ExpectedCount := 0;
ActualCount	  := Sink.LinesWritten;
Test.AssertEqual(ExpectedCount, ActualCount, 'nothing was written');

// Seen but not narrated - the distinction that makes the quiet default safe.
ExpectedCount := 2;
ActualCount	  := Sink.TestsSeen;
Test.AssertEqual(ExpectedCount, ActualCount, 'but both were seen');
Run := TRUE;
END_METHOD

END_FUNCTION_BLOCK

// ---- Tests/LogReporter/TEST_LogReporterWritesFailuresAndErrors.TcPOU
// A failure is an error: the code under test was shown to be wrong. An error is a

// warning: the test could not run, so nothing was shown about the code at all.

//

// Counted apart because a build should react differently to each.//

// WHAT THIS CANNOT CHECK: whether the line actually reached the TwinCAT log, or

// what it says. ADSLOGSTR gives no answer back. The counters prove which BRANCH

// was taken; the wording has to be read once, by eye, in the Logged Events window.

// Saying so is better than a test that implies more than it establishes.
FUNCTION_BLOCK TEST_LogReporterWritesFailuresAndErrors IMPLEMENTS I_Test
VAR
	Sink		  : TestLogReporter;
	ExpectedCount : UDINT;
	ActualCount	  : UDINT;
END_VAR

METHOD Run : BOOL
VAR_INPUT
	Enable : BOOL;
	Test   : I_TestAssertions;
END_VAR
Sink.TestFinished(SuiteLabel	:= 'suite',
				  TestLabel		:= 'a failure',
				  Location		:= '',
				  Status		:= E_TestStatus.Failed,
				  Kind			:= E_FailureKind.ValueMismatch,
				  Summary		:= 'expected 1, actual 2',
				  ElapsedTime	:= 0.0,
				  ElapsedCycles := 1,
				  Assertions	:= 1);

Sink.TestFinished(SuiteLabel	:= 'suite',
				  TestLabel		:= 'an error',
				  Location		:= '',
				  Status		:= E_TestStatus.Errored,
				  Kind			:= E_FailureKind.Environment,
				  Summary		:= 'the axis would not power',
				  ElapsedTime	:= 0.0,
				  ElapsedCycles := 1,
				  Assertions	:= 1);

ExpectedCount := 1;
ActualCount	  := Sink.FailuresLogged;
Test.AssertEqual(ExpectedCount, ActualCount, 'the failure was logged');
ActualCount := Sink.ErrorsLogged;
Test.AssertEqual(ExpectedCount, ActualCount, 'the error was logged separately');
ExpectedCount := 2;
ActualCount	  := Sink.LinesWritten;
Test.AssertEqual(ExpectedCount, ActualCount, 'two lines, not one and not three');
Run := TRUE;
END_METHOD

END_FUNCTION_BLOCK

// ---- Tests/LogReporter/TEST_LogReporterNarratesWhenAsked.TcPOU
// SetVerbosity(TRUE) turns the narration back on, for a rig where the log IS the

// artifact and a passing test that stops appearing is the signal.//

// WHAT THIS CANNOT CHECK: whether the line actually reached the TwinCAT log, or

// what it says. ADSLOGSTR gives no answer back. The counters prove which BRANCH

// was taken; the wording has to be read once, by eye, in the Logged Events window.

// Saying so is better than a test that implies more than it establishes.
FUNCTION_BLOCK TEST_LogReporterNarratesWhenAsked IMPLEMENTS I_Test
VAR
	Sink		  : TestLogReporter;
	ExpectedCount : UDINT;
	ActualCount	  : UDINT;
END_VAR

METHOD Run : BOOL
VAR_INPUT
	Enable : BOOL;
	Test   : I_TestAssertions;
END_VAR
Sink.SetVerbosity(TRUE);
Sink.TestFinished(SuiteLabel	:= 'suite',
				  TestLabel		:= 'a pass',
				  Location		:= '',
				  Status		:= E_TestStatus.Passed,
				  Kind			:= E_FailureKind.None,
				  Summary		:= '',
				  ElapsedTime	:= 0.0,
				  ElapsedCycles := 1,
				  Assertions	:= 1);

ExpectedCount := 1;
ActualCount	  := Sink.LinesWritten;
Test.AssertEqual(ExpectedCount, ActualCount, 'the pass was narrated');

// And it can be turned off again.
Sink.SetVerbosity(FALSE);
Sink.TestFinished(SuiteLabel	:= 'suite',
				  TestLabel		:= 'another pass',
				  Location		:= '',
				  Status		:= E_TestStatus.Passed,
				  Kind			:= E_FailureKind.None,
				  Summary		:= '',
				  ElapsedTime	:= 0.0,
				  ElapsedCycles := 1,
				  Assertions	:= 1);

ActualCount := Sink.LinesWritten;
Test.AssertEqual(ExpectedCount, ActualCount, 'and quiet again afterwards');
Run := TRUE;
END_METHOD

END_FUNCTION_BLOCK

// ---- Tests/LogReporter/TEST_LogReporterAlwaysWritesFrameworkErrors.TcPOU
// A framework error is never silent and is never affected by verbosity. It is the

// framework saying it could not do something - a rejected registration, a teardown

// that overran - and none of those is a test result that can be suppressed.//

// WHAT THIS CANNOT CHECK: whether the line actually reached the TwinCAT log, or

// what it says. ADSLOGSTR gives no answer back. The counters prove which BRANCH

// was taken; the wording has to be read once, by eye, in the Logged Events window.

// Saying so is better than a test that implies more than it establishes.
FUNCTION_BLOCK TEST_LogReporterAlwaysWritesFrameworkErrors IMPLEMENTS I_Test
VAR
	Sink		  : TestLogReporter;
	Fanout		  : TestReporterFanout;
	Attached	  : BOOL;
	ExpectedCount : UDINT;
	ActualCount	  : UDINT;
END_VAR

METHOD Run : BOOL
VAR_INPUT
	Enable : BOOL;
	Test   : I_TestAssertions;
END_VAR
// Quiet mode is the default, and must not silence this.
Sink.FrameworkError(Source := 'a suite', Message := 'registration was rejected');
ExpectedCount := 1;
ActualCount	  := Sink.FrameworkErrorsLogged;
Test.AssertEqual(ExpectedCount, ActualCount, 'logged despite the quiet default');
ActualCount := Sink.LinesWritten;
Test.AssertEqual(ExpectedCount, ActualCount, 'and it produced a line');

// It is a real I_TestReporter, so the fan-out takes it like any other sink.
Attached := Fanout.Attach(Sink);
Test.AssertTrue(Attached, 'the fan-out accepts it');
Fanout.FrameworkError(Source := 'a suite', Message := 'through the fan-out');
ExpectedCount := 2;
ActualCount	  := Sink.FrameworkErrorsLogged;
Test.AssertEqual(ExpectedCount, ActualCount, 'and reaches it that way too');

// Nothing asynchronous, so it never holds a run open.
Test.AssertTrue(Sink.IsIdle, 'the log sink is always idle');
Test.AssertTrue(Fanout.IsIdle, 'so the fan-out is too');
Run := TRUE;
END_METHOD

END_FUNCTION_BLOCK

// ---- Tests/LogReporter/TEST_LogReporterSummarisesASuite.TcPOU
// One line per suite, carrying the counts, with severity following the outcome -

// so a log filtered to errors still shows WHICH suite was responsible rather than

// only the individual failures.//

// WHAT THIS CANNOT CHECK: whether the line actually reached the TwinCAT log, or

// what it says. ADSLOGSTR gives no answer back. The counters prove which BRANCH

// was taken; the wording has to be read once, by eye, in the Logged Events window.

// Saying so is better than a test that implies more than it establishes.
FUNCTION_BLOCK TEST_LogReporterSummarisesASuite IMPLEMENTS I_Test
VAR
	Sink		  : TestLogReporter;
	Tally		  : TestRunTally;
	ExpectedCount : UDINT;
	ActualCount	  : UDINT;
END_VAR

METHOD Run : BOOL
VAR_INPUT
	Enable : BOOL;
	Test   : I_TestAssertions;
END_VAR
Tally.SetLabel('a suite');
Tally.Begin(3);
Tally.Record(Verdict := E_TestStatus.Passed, ElapsedTime := 0.1);
Tally.Record(Verdict := E_TestStatus.Failed, ElapsedTime := 0.1);
Tally.Record(Verdict := E_TestStatus.Skipped, ElapsedTime := 0.0);
Tally.Finish();
Sink.SuiteFinished(Tally);
ExpectedCount := 1;
ActualCount	  := Sink.SuitesSeen;
Test.AssertEqual(ExpectedCount, ActualCount, 'the suite was summarised');
ActualCount := Sink.LinesWritten;
Test.AssertEqual(ExpectedCount, ActualCount, 'in exactly one line');

// A null status is refused rather than dereferenced.
Sink.SuiteFinished(0);
ActualCount := Sink.SuitesSeen;
Test.AssertEqual(ExpectedCount, ActualCount, 'a null status is ignored, not fatal');
Run := TRUE;
END_METHOD

END_FUNCTION_BLOCK

// ---- Tests/LogReporter/TEST_LogReporterNarratesSkipsOnlyWhenAsked.TcPOU
// A skipped test is narrated like a pass - only when asked - and is never counted
// as a failure or an error.
//
// WHAT THIS CANNOT CHECK is the word on the line. It now reads "skipped", where the
// pass branch it used to share would have written "passed"; ADSLOGSTR gives no
// answer back, so the counters prove which BRANCH was taken and the wording has to
// be read once, by eye, in the Logged Events window - the same limit
// TEST_LogReporterNarratesWhenAsked states.
//
// It therefore passed before skipped verdicts reached sinks as well as after. It
// is kept as the guard on the branch: a skip routed into the failure or error
// branch, or logged when narration is off, turns it red.
FUNCTION_BLOCK TEST_LogReporterNarratesSkipsOnlyWhenAsked IMPLEMENTS I_Test
VAR
	Sink		  : TestLogReporter;
	ExpectedCount : UDINT;
	ActualCount	  : UDINT;
END_VAR

METHOD Run : BOOL
VAR_INPUT
	Enable : BOOL;
	Test   : I_TestAssertions;
END_VAR
Sink.TestFinished(SuiteLabel	:= 'suite',
				  TestLabel		:= 'a skipped test',
				  Location		:= '',
				  Status		:= E_TestStatus.Skipped,
				  Kind			:= E_FailureKind.None,
				  Summary		:= '',
				  ElapsedTime	:= 0.0,
				  ElapsedCycles := 0,
				  Assertions	:= 0);
ExpectedCount := 0;
ActualCount	  := Sink.LinesWritten;
Test.AssertEqual(ExpectedCount, ActualCount, 'quiet about a skip by default');

Sink.SetVerbosity(TRUE);
Sink.TestFinished(SuiteLabel	:= 'suite',
				  TestLabel		:= 'another skipped test',
				  Location		:= '',
				  Status		:= E_TestStatus.Skipped,
				  Kind			:= E_FailureKind.None,
				  Summary		:= '',
				  ElapsedTime	:= 0.0,
				  ElapsedCycles := 0,
				  Assertions	:= 0);
ExpectedCount := 1;
ActualCount	  := Sink.LinesWritten;
Test.AssertEqual(ExpectedCount, ActualCount, 'narrated in one line when asked');

ExpectedCount := 0;
ActualCount	  := Sink.FailuresLogged;
Test.AssertEqual(ExpectedCount, ActualCount, 'never as a failure');
ActualCount := Sink.ErrorsLogged;
Test.AssertEqual(ExpectedCount, ActualCount, 'nor as an error');
Run := TRUE;
END_METHOD

END_FUNCTION_BLOCK

// ---- Tests/LogReporter/TEST_LogReporterNamesASkippedAndAnErroredRun.TcPOU
// A skipped run and an errored run each get a banner of their own, at the severity
// the suite line uses: RUN SKIPPED as a message, RUN ERRORED as an error.
//
// Until the run banner copied the suite line's four branches, both printed RUN
// FAILED at error severity - so a run that exercised nothing turned an error-filtered
// log red, and a run that could not be trusted read as a defect in the code.
//
// WHAT THIS CANNOT CHECK: the word on the line, or its severity. ADSLOGSTR gives no
// answer back. The counters prove each banner was written between its two rules;
// the wording is read by eye, and this test exists so that every verifier log has
// both banners in it to read. They carry the prefix 'verifier sample - ' and name
// themselves as samples: RUN ERRORED is an error-severity line on every run, and must
// not be taken for this run's result.
FUNCTION_BLOCK TEST_LogReporterNamesASkippedAndAnErroredRun IMPLEMENTS I_Test
VAR
	Sink	   : TestLogReporter;
	SkippedRun : TestRunTally;
	ErroredRun : TestRunTally;

	ExpectedCount	: UDINT;
	ActualCount		: UDINT;
	ExpectedOutcome : E_RunOutcome;
	ActualOutcome	: E_RunOutcome;
END_VAR

METHOD Run : BOOL
VAR_INPUT
	Enable : BOOL;
	Test   : I_TestAssertions;
END_VAR
Sink.SetPrefix('verifier sample - ');

// Two runs built by hand, and checked before they are logged: a banner is only
// worth reading if the outcome behind it is the one intended.
SkippedRun.SetLabel('a skipped run');
SkippedRun.Begin(2);
SkippedRun.Record(Verdict := E_TestStatus.Skipped, ElapsedTime := 0.0);
SkippedRun.Record(Verdict := E_TestStatus.Skipped, ElapsedTime := 0.0);
SkippedRun.Finish();
ExpectedOutcome := E_RunOutcome.Skipped;
ActualOutcome	:= SkippedRun.Outcome;
Test.AssertEqual(ExpectedOutcome, ActualOutcome, 'the first sample run is Skipped');

ErroredRun.SetLabel('an errored run');
ErroredRun.Begin(2);
ErroredRun.Record(Verdict := E_TestStatus.Passed, ElapsedTime := 0.1);
ErroredRun.Record(Verdict := E_TestStatus.Errored, ElapsedTime := 0.1);
ErroredRun.Finish();
ExpectedOutcome := E_RunOutcome.Errored;
ActualOutcome	:= ErroredRun.Outcome;
Test.AssertEqual(ExpectedOutcome, ActualOutcome, 'the second is Errored');

// Expect, in the Logged Events window:
//   verifier sample - ===  RUN SKIPPED 0 passed, 0 failed, 0 errored, 2 skipped, of 2 ...  (Message)
//   verifier sample - ===  RUN ERRORED 1 passed, 0 failed, 1 errored, 0 skipped, of 2 ...  (Error)
Sink.RunFinished(Status := SkippedRun, TargetInfo := 'a sample, not this run');
ExpectedCount := 3;
ActualCount	  := Sink.LinesWritten;
Test.AssertEqual(ExpectedCount, ActualCount, 'the skipped run got a banner between two rules');

Sink.RunFinished(Status := ErroredRun, TargetInfo := 'a sample, not this run');
ExpectedCount := 6;
ActualCount	  := Sink.LinesWritten;
Test.AssertEqual(ExpectedCount, ActualCount, 'and so did the errored run');

// A null status is refused rather than dereferenced.
Sink.RunFinished(Status := 0, TargetInfo := '');
ActualCount := Sink.LinesWritten;
Test.AssertEqual(ExpectedCount, ActualCount, 'a null status writes nothing');
Run := TRUE;
END_METHOD

END_FUNCTION_BLOCK

// ---- Tests/JUnitReporter/TEST_JUnitReporterOpensOnRunStarted.TcPOU
// The document is opened by RunStarted, not inferred from the first result.

//

// Proved by driving a run whose ONLY content is a framework error - no test and no

// suite - so nothing but RunStarted could have opened the document.

//

// LENGTHS ARE COMPARED, NOT TESTED AGAINST ZERO. An untouched FB_XmlDomParser

// already holds a minimal document, so "no document" is not "no length", and

// pinning the exact figure would be testing Beckhoff's implementation rather than

// this one.
FUNCTION_BLOCK TEST_JUnitReporterOpensOnRunStarted IMPLEMENTS I_Test
VAR
	Writer : TestJUnitReporter;
	Spy	   : SpyReporter;

	// Captured rather than assumed. The baseline is whatever an untouched parser

	// happens to hold, and pinning that number would be testing Beckhoff's

	// implementation rather than this one.
	Baseline	  : UDINT;
	Opened		  : UDINT;
	Length		  : UDINT;
	ExpectedCount : UDINT;
	ActualCount	  : UDINT;
END_VAR

METHOD Run : BOOL
VAR_INPUT
	Enable : BOOL;
	Test   : I_TestAssertions;
END_VAR
Writer.AttachErrorSink(Spy);

// Whatever an untouched parser holds.
Baseline := Writer.DocumentLength;
Writer.RunStarted(Label := 'a run', TargetInfo := 'a target');

// Opened: it now carries structure, if not yet results.
Opened := Writer.DocumentLength;
Test.AssertTrue(Opened > Baseline, 'RunStarted opened the document');
Writer.FrameworkError(Source := 'somewhere', Message := 'something went wrong');
Length := Writer.DocumentLength;
Test.AssertTrue(Length > Opened, 'and a framework error is recorded in it, with no test involved');
Run := TRUE;
END_METHOD

END_FUNCTION_BLOCK

// ---- Tests/EventReporter/TEST_EventReporterSendsAndDoesNotFail.TcPOU
// The load-bearing test for this sink: an event was accepted by the EventLogger,

// and no call returned a failing HRESULT.

//

// FailedSends is what distinguishes "the event class is not registered" from

// "everything is fine" - both look identical from the PLC otherwise, because a

// failed Create produces exactly as much visible output as a successful one that

// nobody is watching.
FUNCTION_BLOCK TEST_EventReporterSendsAndDoesNotFail IMPLEMENTS I_Test
VAR
	Sink		  : TestEventReporter;
	ExpectedCount : UDINT;
	ActualCount	  : UDINT;
	Error		  : HRESULT;
END_VAR

METHOD Run : BOOL
VAR_INPUT
	Enable : BOOL;
	Test   : I_TestAssertions;
END_VAR
Sink.TestFinished(SuiteLabel	:= 'suite',
				  TestLabel		:= 'a failure',
				  Location		:= '',
				  Status		:= E_TestStatus.Failed,
				  Kind			:= E_FailureKind.ValueMismatch,
				  Summary		:= 'expected 1, actual 2',
				  ElapsedTime	:= 0.0,
				  ElapsedCycles := 1,
				  Assertions	:= 1);

ExpectedCount := 1;
ActualCount	  := Sink.EventsSent;
Test.AssertEqual(ExpectedCount, ActualCount, 'the event was accepted');
ExpectedCount := 0;
ActualCount	  := Sink.FailedSends;
Test.AssertEqual(ExpectedCount, ActualCount, 'and nothing was refused');

// Reported rather than swallowed. If this is non-zero the HRESULT says why.
Error := Sink.LastError;
Test.AssertTrue(Error = 0, 'no HRESULT was returned');
Run := TRUE;
END_METHOD

END_FUNCTION_BLOCK

// ---- Tests/EventReporter/TEST_EventReporterIsQuietAboutPasses.TcPOU
// Quiet by default. Eighty Info events bury the two Errors, and the counts are

// already available through I_TestRunStatus for anyone who wants them.

//

// The Verbose severity exists for narration and is filtered out of most views

// anyway - but not raising the event at all is cheaper still.
FUNCTION_BLOCK TEST_EventReporterIsQuietAboutPasses IMPLEMENTS I_Test
VAR
	Sink		  : TestEventReporter;
	ExpectedCount : UDINT;
	ActualCount	  : UDINT;
END_VAR

METHOD Run : BOOL
VAR_INPUT
	Enable : BOOL;
	Test   : I_TestAssertions;
END_VAR
Sink.TestFinished(SuiteLabel	:= 'suite',
				  TestLabel		:= 'a pass',
				  Location		:= '',
				  Status		:= E_TestStatus.Passed,
				  Kind			:= E_FailureKind.None,
				  Summary		:= '',
				  ElapsedTime	:= 0.0,
				  ElapsedCycles := 1,
				  Assertions	:= 1);

ExpectedCount := 0;
ActualCount	  := Sink.EventsSent;
Test.AssertEqual(ExpectedCount, ActualCount, 'nothing was raised');
Sink.SetVerbosity(TRUE);
Sink.TestFinished(SuiteLabel	:= 'suite',
				  TestLabel		:= 'a pass',
				  Location		:= '',
				  Status		:= E_TestStatus.Passed,
				  Kind			:= E_FailureKind.None,
				  Summary		:= '',
				  ElapsedTime	:= 0.0,
				  ElapsedCycles := 1,
				  Assertions	:= 1);

ExpectedCount := 1;
ActualCount	  := Sink.EventsSent;
Test.AssertEqual(ExpectedCount, ActualCount, 'and narration turns it on');
ExpectedCount := 0;
ActualCount	  := Sink.FailedSends;
Test.AssertEqual(ExpectedCount, ActualCount, 'the Verbose event was accepted too');
Run := TRUE;
END_METHOD

END_FUNCTION_BLOCK

// ---- Tests/EventReporter/TEST_EventReporterRaisesEachOutcomeOnce.TcPOU
// One event per notification, whatever the outcome - failures, errors, suite

// results and framework errors all raise exactly one.

//

// The IDs and severities differ per outcome so a filtered view can show suite

// results without every individual failure; what this checks is that each path

// reaches the logger and none raises twice.
FUNCTION_BLOCK TEST_EventReporterRaisesEachOutcomeOnce IMPLEMENTS I_Test
VAR
	Sink		  : TestEventReporter;
	Tally		  : TestRunTally;
	ExpectedCount : UDINT;
	ActualCount	  : UDINT;
END_VAR

METHOD Run : BOOL
VAR_INPUT
	Enable : BOOL;
	Test   : I_TestAssertions;
END_VAR
Sink.TestFinished(SuiteLabel	:= 's',
				  TestLabel		:= 'failed',
				  Location		:= '',
				  Status		:= E_TestStatus.Failed,
				  Kind			:= E_FailureKind.ValueMismatch,
				  Summary		:= 'x',
				  ElapsedTime	:= 0.0,
				  ElapsedCycles := 1,
				  Assertions	:= 1);

Sink.TestFinished(SuiteLabel	:= 's',
				  TestLabel		:= 'errored',
				  Location		:= '',
				  Status		:= E_TestStatus.Errored,
				  Kind			:= E_FailureKind.Environment,
				  Summary		:= 'y',
				  ElapsedTime	:= 0.0,
				  ElapsedCycles := 1,
				  Assertions	:= 1);

Sink.FrameworkError(Source := 's', Message := 'something the framework could not do');
Tally.SetLabel('s');
Tally.Begin(2);
Tally.Record(Verdict := E_TestStatus.Passed, ElapsedTime := 0.1);
Tally.Record(Verdict := E_TestStatus.Failed, ElapsedTime := 0.1);
Tally.Finish();
Sink.SuiteFinished(Tally);
Sink.RunFinished(Status := Tally, TargetInfo := 'the verifier');
ExpectedCount := 5;
ActualCount	  := Sink.EventsSent;
Test.AssertEqual(ExpectedCount, ActualCount, 'five notifications, five events');
ExpectedCount := 0;
ActualCount	  := Sink.FailedSends;
Test.AssertEqual(ExpectedCount, ActualCount, 'none refused');

// A null status is refused rather than dereferenced, and raises nothing.
Sink.SuiteFinished(0);
Sink.RunFinished(Status := 0, TargetInfo := '');
ExpectedCount := 5;
ActualCount	  := Sink.EventsSent;
Test.AssertEqual(ExpectedCount, ActualCount, 'a null status raises nothing');
Run := TRUE;
END_METHOD

END_FUNCTION_BLOCK

// ---- Tests/EventReporter/TEST_EventReporterWorksThroughTheFanout.TcPOU
// It is an ordinary I_TestReporter, so the fan-out takes it beside any other sink

// and both receive everything.

//

// Also the case that matters for a build: the ADSLOGSTR sink and the EventLogger

// sink attached together, because they answer different questions and a rig

// usually wants both.
FUNCTION_BLOCK TEST_EventReporterWorksThroughTheFanout IMPLEMENTS I_Test
VAR
	Fanout		  : TestReporterFanout;
	Events		  : TestEventReporter;
	LogSink		  : TestLogReporter;
	Attached	  : BOOL;
	ExpectedCount : UDINT;
	ActualCount	  : UDINT;
END_VAR

METHOD Run : BOOL
VAR_INPUT
	Enable : BOOL;
	Test   : I_TestAssertions;
END_VAR
Attached := Fanout.Attach(Events) AND Fanout.Attach(LogSink);
Test.AssertTrue(Attached, 'both sinks attached');
Fanout.FrameworkError(Source := 'the fan-out', Message := 'reached both sinks');
ExpectedCount := 1;
ActualCount	  := Events.EventsSent;
Test.AssertEqual(ExpectedCount, ActualCount, 'the event sink raised one');
ActualCount := LogSink.FrameworkErrorsLogged;
Test.AssertEqual(ExpectedCount, ActualCount, 'and the log sink wrote one');

// Neither starts asynchronous work, so a run is never held open by them.
Test.AssertTrue(Events.IsIdle, 'the event sink is idle');
Test.AssertTrue(Fanout.IsIdle, 'so the fan-out is');

// Suspending covers both, which is what makes an individual re-run silent.
Fanout.Suspend();
Fanout.FrameworkError(Source := 'the fan-out', Message := 'must not be raised');
ActualCount := Events.EventsSent;
Test.AssertEqual(ExpectedCount, ActualCount, 'and Suspend silences it too');
Run := TRUE;
END_METHOD

END_FUNCTION_BLOCK

// ---- Tests/EventReporter/TEST_EventReporterDoesNotCallASkipAPass.TcPOU
// A skipped test raises no event, even with narration on - and above all not
// TestPassed.
//
// The event class has one per-test event for each of Passed, Failed and Errored,
// and none for Skipped. Narration once sent every verdict that was not a failure
// or an error down the pass branch, which was harmless while no skipped verdict
// ever reached a sink. Once one does, an operator filtering for passes would see a
// test that never ran reported as one that did.
//
// The skip is not lost: the suite's own SuiteSkipped event carries the count. A
// per-test skipped event needs an entry in the event class first.
//
// Asserts FailedSends as well as EventsSent, so this holds whether or not the
// event class is registered on the target: nothing may even be attempted.
FUNCTION_BLOCK TEST_EventReporterDoesNotCallASkipAPass IMPLEMENTS I_Test
VAR
	Sink		  : TestEventReporter;
	ExpectedCount : UDINT;
	ActualCount	  : UDINT;
END_VAR

METHOD Run : BOOL
VAR_INPUT
	Enable : BOOL;
	Test   : I_TestAssertions;
END_VAR
Sink.SetVerbosity(TRUE);
Sink.TestFinished(SuiteLabel	:= 'suite',
				  TestLabel		:= 'a skipped test',
				  Location		:= '',
				  Status		:= E_TestStatus.Skipped,
				  Kind			:= E_FailureKind.None,
				  Summary		:= '',
				  ElapsedTime	:= 0.0,
				  ElapsedCycles := 0,
				  Assertions	:= 0);
ExpectedCount := 0;
ActualCount	  := Sink.EventsSent;
Test.AssertEqual(ExpectedCount, ActualCount, 'a skipped test raised no event, even with narration on');
ActualCount := Sink.FailedSends;
Test.AssertEqual(ExpectedCount, ActualCount, 'and none was even attempted');

// Narration really is on: a pass still raises one. Without this, a sink that had
// simply stopped narrating would pass the checks above.
Sink.TestFinished(SuiteLabel	:= 'suite',
				  TestLabel		:= 'a pass',
				  Location		:= '',
				  Status		:= E_TestStatus.Passed,
				  Kind			:= E_FailureKind.None,
				  Summary		:= '',
				  ElapsedTime	:= 0.0,
				  ElapsedCycles := 0,
				  Assertions	:= 0);
ExpectedCount := 1;
ActualCount	  := Sink.EventsSent + Sink.FailedSends;
Test.AssertEqual(ExpectedCount, ActualCount, 'while a pass is still narrated');
Run := TRUE;
END_METHOD

END_FUNCTION_BLOCK

// ---- Tests/EventReporter/TEST_EventReporterNamesASkippedAndAnErroredRun.TcPOU
// A skipped run raises RunSkipped and an errored run raises RunErrored, and the
// logger accepts both.
//
// The run once had two events: RunPassed, and RunFailed for everything else. So a
// run that exercised nothing raised an Error-severity RunFailed, and a run that
// could not be trusted read as a defect in the code. RunSkipped (Info) and
// RunErrored (Error) were added to the event class to match the suite's four.
//
// WHAT THIS CAN CHECK: that each run raised exactly one event and the logger
// refused none. It does NOT prove the class on the target carries RunSkipped and
// RunErrored: whether the logger refuses an event its class does not define is not
// established. That proof is the library compiling at all, since the reporter
// names both.
//
// WHAT IT CANNOT: which event was raised. Read that in the logger. RunSkipped is
// Info and stands apart; RunErrored shares Error severity and text form with
// RunFailed, so tell those two apart by event ID - 13 against 7.
FUNCTION_BLOCK TEST_EventReporterNamesASkippedAndAnErroredRun IMPLEMENTS I_Test
VAR
	Sink	   : TestEventReporter;
	SkippedRun : TestRunTally;
	ErroredRun : TestRunTally;

	ExpectedCount	: UDINT;
	ActualCount		: UDINT;
	ExpectedOutcome : E_RunOutcome;
	ActualOutcome	: E_RunOutcome;
END_VAR

METHOD Run : BOOL
VAR_INPUT
	Enable : BOOL;
	Test   : I_TestAssertions;
END_VAR
// Two runs built by hand, and checked before they are raised.
SkippedRun.SetLabel('a skipped run');
SkippedRun.Begin(2);
SkippedRun.Record(Verdict := E_TestStatus.Skipped, ElapsedTime := 0.0);
SkippedRun.Record(Verdict := E_TestStatus.Skipped, ElapsedTime := 0.0);
SkippedRun.Finish();
ExpectedOutcome := E_RunOutcome.Skipped;
ActualOutcome	:= SkippedRun.Outcome;
Test.AssertEqual(ExpectedOutcome, ActualOutcome, 'the first sample run is Skipped');

ErroredRun.SetLabel('an errored run');
ErroredRun.Begin(2);
ErroredRun.Record(Verdict := E_TestStatus.Passed, ElapsedTime := 0.1);
ErroredRun.Record(Verdict := E_TestStatus.Errored, ElapsedTime := 0.1);
ErroredRun.Finish();
ExpectedOutcome := E_RunOutcome.Errored;
ActualOutcome	:= ErroredRun.Outcome;
Test.AssertEqual(ExpectedOutcome, ActualOutcome, 'the second is Errored');

// Named as samples, so neither is taken for this run's result.
Sink.RunFinished(Status := SkippedRun, TargetInfo := 'a sample, not this run');
Sink.RunFinished(Status := ErroredRun, TargetInfo := 'a sample, not this run');

ExpectedCount := 2;
ActualCount	  := Sink.EventsSent;
Test.AssertEqual(ExpectedCount, ActualCount, 'each sample run raised one event');
ExpectedCount := 0;
ActualCount	  := Sink.FailedSends;
Test.AssertEqual(ExpectedCount, ActualCount, 'and the logger refused neither');

// A null status is refused rather than dereferenced.
Sink.RunFinished(Status := 0, TargetInfo := '');
ExpectedCount := 2;
ActualCount	  := Sink.EventsSent + Sink.FailedSends;
Test.AssertEqual(ExpectedCount, ActualCount, 'a null status raises nothing');
Run := TRUE;
END_METHOD

END_FUNCTION_BLOCK

// ---- Tests/JUnitReporter/TEST_JUnitReporterWritesTheDocument.TcPOU
// The document reaches disk, and the write reports success.

//

// It also checks the document is NOT EMPTY, which FilesWritten alone cannot say.

// A successful write of a bare XML declaration looks identical to a successful

// write of a full document - and that is exactly what happened the first time

// this ran: 23 bytes, no error, everything apparently fine.

//

// WHAT THIS STILL CANNOT CHECK: whether the XML is well formed or whether CI can

// parse it. Nothing in the PLC reads the file back. Open it once, by eye.

//

// Writes to the 4026 boot folder. If that path is wrong for this machine the test

// fails as a write failure, which is the correct outcome and not a false alarm.
FUNCTION_BLOCK TEST_JUnitReporterWritesTheDocument IMPLEMENTS I_Test
VAR
	Writer		  : TestJUnitReporter;
	Spy			  : SpyReporter;
	Tally		  : TestRunTally;
	Phase		  : DINT;
	Scans		  : DINT;
	Path		  : T_MaxString := 'C:\ProgramData\Beckhoff\TwinCAT\3.1\Boot\TestHarnessCoreVerifier.xml';
	ExpectedCount : UDINT;
	ActualCount	  : UDINT;
	Error		  : HRESULT;
	Length		  : UDINT;
END_VAR

METHOD Run : BOOL
VAR_INPUT
	Enable : BOOL;
	Test   : I_TestAssertions;
END_VAR
Scans := Scans + 1;
IF Scans > 2000 THEN
	Test.Fail('the write never finished');
	Run := TRUE;
	RETURN;
END_IF

CASE Phase OF
	0:
		Writer.SetPath(Path);
		Writer.AttachErrorSink(Spy);
		Tally.SetLabel('a suite');
		Tally.Begin(1);
		Writer.TestStarted(SuiteLabel := 'a suite', TestLabel := 'a test', Location := 'Verifier.Somewhere');
		Writer.CheckPassed(StepLabel := '', Detail := '');
		Writer.CheckFailed(StepLabel  := 'Home',
						   Kind		  := E_FailureKind.ValueMismatch,
						   Expected	  := '1',
						   Actual	  := '2',
						   Diagnostic := 'expected 1, actual 2',
						   Message	  := 'deliberate');

		Writer.TestFinished(SuiteLabel	  := 'a suite',
							TestLabel	  := 'a test',
							Location	  := 'Verifier.Somewhere',
							Status		  := E_TestStatus.Failed,
							Kind		  := E_FailureKind.ValueMismatch,
							Summary		  := 'Home: expected 1, actual 2 - deliberate',
							ElapsedTime	  := 0.01,
							ElapsedCycles := 1,
							Assertions	  := 2);

		Tally.Record(Verdict := E_TestStatus.Failed, ElapsedTime := 0.01);
		Tally.Finish();
		Writer.SuiteFinished(Tally);
		Writer.RunFinished(Status := Tally, TargetInfo := 'the verifier');
		Phase := 1;
		Run	  := FALSE;

	1:
		// The write is asynchronous. This is what CyclicLogic exists for.
		Writer.CyclicLogic();
		IF Writer.IsIdle THEN
			Phase := 2;
		END_IF

		Run := FALSE;

	2:
		ExpectedCount := 1;
		ActualCount	  := Writer.FilesWritten;
		Test.AssertEqual(ExpectedCount, ActualCount, 'the document was written');
		ExpectedCount := 0;
		ActualCount	  := Writer.WriteFailures;
		Test.AssertEqual(ExpectedCount, ActualCount, 'with no failures');
		Error := Writer.LastError;
		Test.AssertTrue(Error = 0, 'and no HRESULT');

		// The bar is deliberately well above the 23 bytes an empty document produces,

		// and well below what this run actually generates. It is a smoke test for

		// "something was built", not an assertion about the exact bytes.
		Length := Writer.DocumentLength;
		Test.AssertTrue(Length > 200, 'the document has real content in it');

		// A failed write raises a framework error. A successful one must not.
		ExpectedCount := 0;
		ActualCount	  := Spy.FrameworkErrorCalls;
		Test.AssertEqual(ExpectedCount, ActualCount, 'nothing was reported as wrong');
		Run := TRUE;
END_CASE
END_METHOD

END_FUNCTION_BLOCK

// ---- Tests/JUnitReporter/TEST_JUnitReporterIsBusyWhileWriting.TcPOU
// The ONLY sink where IsIdle means anything. Every other one returns TRUE

// constantly because nothing they do outlives the call.

//

// CI must wait for this as well as IsComplete: a run finishing and its document

// reaching disk are different events, and copying between them yields a truncated

// artifact - which reads as a broken pipeline rather than a finished run.

//

// A fast local write could hide a missing IsIdle. Checking it on the scan the

// write is REQUESTED, before CyclicLogic has run at all, is what makes this test

// mean something.
FUNCTION_BLOCK TEST_JUnitReporterIsBusyWhileWriting IMPLEMENTS I_Test
VAR
	Writer		  : TestJUnitReporter;
	Spy			  : SpyReporter;
	Tally		  : TestRunTally;
	Phase		  : DINT;
	Scans		  : DINT;
	Path		  : T_MaxString := 'C:\ProgramData\Beckhoff\TwinCAT\3.1\Boot\TestHarnessCoreVerifier_Busy.xml';
	IdleAtStart	  : BOOL;
	IdleWhenAsked : BOOL;
	IdleAtEnd	  : BOOL;
	ExpectedCount : UDINT;
	ActualCount	  : UDINT;
END_VAR

METHOD Run : BOOL
VAR_INPUT
	Enable : BOOL;
	Test   : I_TestAssertions;
END_VAR
Scans := Scans + 1;
IF Scans > 2000 THEN
	Test.Fail('the write never finished');
	Run := TRUE;
	RETURN;
END_IF

CASE Phase OF
	0:
		Writer.SetPath(Path);
		IdleAtStart := Writer.IsIdle;
		Writer.AttachErrorSink(Spy);
		Tally.SetLabel('a suite');
		Tally.Begin(1);
		Writer.TestStarted(SuiteLabel := 'a suite', TestLabel := 'a test', Location := 'Verifier.Somewhere');
		Writer.CheckPassed(StepLabel := '', Detail := '');
		Writer.CheckFailed(StepLabel  := 'Home',
						   Kind		  := E_FailureKind.ValueMismatch,
						   Expected	  := '1',
						   Actual	  := '2',
						   Diagnostic := 'expected 1, actual 2',
						   Message	  := 'deliberate');

		Writer.TestFinished(SuiteLabel	  := 'a suite',
							TestLabel	  := 'a test',
							Location	  := 'Verifier.Somewhere',
							Status		  := E_TestStatus.Failed,
							Kind		  := E_FailureKind.ValueMismatch,
							Summary		  := 'Home: expected 1, actual 2 - deliberate',
							ElapsedTime	  := 0.01,
							ElapsedCycles := 1,
							Assertions	  := 2);

		Tally.Record(Verdict := E_TestStatus.Failed, ElapsedTime := 0.01);
		Tally.Finish();
		Writer.SuiteFinished(Tally);
		Writer.RunFinished(Status := Tally, TargetInfo := 'the verifier');

		// Requested, and nothing has driven it yet.
		IdleWhenAsked := Writer.IsIdle;
		Phase		  := 1;
		Run			  := FALSE;

	1:
		Writer.CyclicLogic();
		IF Writer.IsIdle THEN
			IdleAtEnd := TRUE;
			Phase	  := 2;
		END_IF

		Run := FALSE;

	2:
		Test.AssertTrue(IdleAtStart, 'idle before anything was asked of it');
		Test.AssertFalse(IdleWhenAsked, 'NOT idle once the write is requested');
		Test.AssertTrue(IdleAtEnd, 'idle again once the file lands');
		ExpectedCount := 1;
		ActualCount	  := Writer.FilesWritten;
		Test.AssertEqual(ExpectedCount, ActualCount, 'and it really wrote');
		Run := TRUE;
END_CASE
END_METHOD

END_FUNCTION_BLOCK

// ---- Tests/JUnitReporter/TEST_JUnitReporterReportsAFailedWrite.TcPOU
// R3, and the reason this test exists at all.

//

// Discarding the FALSE and the HRESULT from SaveDocumentToFile would make a bad

// path indistinguishable from a suite that never finished. A successful write

// proves nothing about that; only a failing one does.

//

// The path names a folder that does not exist.
FUNCTION_BLOCK TEST_JUnitReporterReportsAFailedWrite IMPLEMENTS I_Test
VAR
	Writer		  : TestJUnitReporter;
	Spy			  : SpyReporter;
	Tally		  : TestRunTally;
	Phase		  : DINT;
	Scans		  : DINT;
	BadPath		  : T_MaxString := 'C:\ProgramData\Beckhoff\TwinCAT\3.1\Boot\NoSuchFolder_TestHarness\r.xml';
	ExpectedCount : UDINT;
	ActualCount	  : UDINT;
	Error		  : HRESULT;
END_VAR

METHOD Run : BOOL
VAR_INPUT
	Enable : BOOL;
	Test   : I_TestAssertions;
END_VAR
Scans := Scans + 1;
IF Scans > 2000 THEN
	Test.Fail('the write never finished');
	Run := TRUE;
	RETURN;
END_IF

CASE Phase OF
	0:
		Writer.SetPath(BadPath);
		Writer.AttachErrorSink(Spy);
		Tally.SetLabel('a suite');
		Tally.Begin(1);
		Writer.TestStarted(SuiteLabel := 'a suite', TestLabel := 'a test', Location := 'Verifier.Somewhere');
		Writer.CheckPassed(StepLabel := '', Detail := '');
		Writer.CheckFailed(StepLabel  := 'Home',
						   Kind		  := E_FailureKind.ValueMismatch,
						   Expected	  := '1',
						   Actual	  := '2',
						   Diagnostic := 'expected 1, actual 2',
						   Message	  := 'deliberate');

		Writer.TestFinished(SuiteLabel	  := 'a suite',
							TestLabel	  := 'a test',
							Location	  := 'Verifier.Somewhere',
							Status		  := E_TestStatus.Failed,
							Kind		  := E_FailureKind.ValueMismatch,
							Summary		  := 'Home: expected 1, actual 2 - deliberate',
							ElapsedTime	  := 0.01,
							ElapsedCycles := 1,
							Assertions	  := 2);

		Tally.Record(Verdict := E_TestStatus.Failed, ElapsedTime := 0.01);
		Tally.Finish();
		Writer.SuiteFinished(Tally);
		Writer.RunFinished(Status := Tally, TargetInfo := 'the verifier');
		Phase := 1;
		Run	  := FALSE;

	1:
		Writer.CyclicLogic();
		IF Writer.IsIdle THEN
			Phase := 2;
		END_IF

		Run := FALSE;

	2:
		ExpectedCount := 0;
		ActualCount	  := Writer.FilesWritten;
		Test.AssertEqual(ExpectedCount, ActualCount, 'nothing was written');
		ExpectedCount := 1;
		ActualCount	  := Writer.WriteFailures;
		Test.AssertEqual(ExpectedCount, ActualCount, 'and the failure was counted');

		// Not swallowed: the HRESULT says WHY.
		Error := Writer.LastError;
		Test.AssertTrue(Error <> 0, 'the HRESULT was kept');

		// And it reached a sink, so the failure is visible without inspecting this

		// object.
		ExpectedCount := 1;
		ActualCount	  := Spy.FrameworkErrorCalls;
		Test.AssertEqual(ExpectedCount, ActualCount, 'and was reported as a framework error');
		Run := TRUE;
END_CASE
END_METHOD

END_FUNCTION_BLOCK

// ---- Tests/JUnitReporter/TEST_JUnitReporterRefusesWithNoPath.TcPOU
// Asking for a write with no path set is a failure, not silence.

//

// It is caught before anything asynchronous starts, so IsIdle never drops - there

// is nothing to wait for.
FUNCTION_BLOCK TEST_JUnitReporterRefusesWithNoPath IMPLEMENTS I_Test
VAR
	Writer		  : TestJUnitReporter;
	Spy			  : SpyReporter;
	Tally		  : TestRunTally;
	Phase		  : DINT;
	Scans		  : DINT;
	ExpectedCount : UDINT;
	ActualCount	  : UDINT;
END_VAR

METHOD Run : BOOL
VAR_INPUT
	Enable : BOOL;
	Test   : I_TestAssertions;
END_VAR
Scans := Scans + 1;
IF Scans > 2000 THEN
	Test.Fail('the write never finished');
	Run := TRUE;
	RETURN;
END_IF

CASE Phase OF
	0:
		// Deliberately no SetPath.
		Writer.AttachErrorSink(Spy);
		Tally.SetLabel('a suite');
		Tally.Begin(1);
		Writer.TestStarted(SuiteLabel := 'a suite', TestLabel := 'a test', Location := 'Verifier.Somewhere');
		Writer.CheckPassed(StepLabel := '', Detail := '');
		Writer.CheckFailed(StepLabel  := 'Home',
						   Kind		  := E_FailureKind.ValueMismatch,
						   Expected	  := '1',
						   Actual	  := '2',
						   Diagnostic := 'expected 1, actual 2',
						   Message	  := 'deliberate');

		Writer.TestFinished(SuiteLabel	  := 'a suite',
							TestLabel	  := 'a test',
							Location	  := 'Verifier.Somewhere',
							Status		  := E_TestStatus.Failed,
							Kind		  := E_FailureKind.ValueMismatch,
							Summary		  := 'Home: expected 1, actual 2 - deliberate',
							ElapsedTime	  := 0.01,
							ElapsedCycles := 1,
							Assertions	  := 2);

		Tally.Record(Verdict := E_TestStatus.Failed, ElapsedTime := 0.01);
		Tally.Finish();
		Writer.SuiteFinished(Tally);
		Writer.RunFinished(Status := Tally, TargetInfo := 'the verifier');
		Phase := 1;
		Run	  := FALSE;

	1:
		Test.AssertTrue(Writer.IsIdle, 'no write was started');
		ExpectedCount := 1;
		ActualCount	  := Writer.WriteFailures;
		Test.AssertEqual(ExpectedCount, ActualCount, 'but it counted as a failure');
		ExpectedCount := 1;
		ActualCount	  := Spy.FrameworkErrorCalls;
		Test.AssertEqual(ExpectedCount, ActualCount, 'and said so');
		ExpectedCount := 0;
		ActualCount	  := Writer.FilesWritten;
		Test.AssertEqual(ExpectedCount, ActualCount, 'and wrote nothing');
		Run := TRUE;
END_CASE
END_METHOD

END_FUNCTION_BLOCK

// ---- Tests/JUnitReporter/TEST_JUnitReporterWritesNothingWhenNothingRan.TcPOU
// A sink that was never part of a run writes nothing.

//

// The distinction is RunStarted. Without it no document was ever opened, so there

// is nothing to write and inventing one would claim something happened.

//

// AN EMPTY RUN IS DIFFERENT and does produce a document, carrying tests="0" - the

// second half of this test. A missing file is ambiguous, because a configuration

// problem and a run with no tests look identical from CI; tests="0" says which.
FUNCTION_BLOCK TEST_JUnitReporterWritesNothingWhenNothingRan IMPLEMENTS I_Test
VAR
	Writer		  : TestJUnitReporter;
	Spy			  : SpyReporter;
	Tally		  : TestRunTally;
	Phase		  : DINT;
	Scans		  : DINT;
	Path		  : T_MaxString := 'C:\ProgramData\Beckhoff\TwinCAT\3.1\Boot\TestHarnessCoreVerifier_Empty.xml';
	ExpectedCount : UDINT;
	ActualCount	  : UDINT;
END_VAR

METHOD Run : BOOL
VAR_INPUT
	Enable : BOOL;
	Test   : I_TestAssertions;
END_VAR
Scans := Scans + 1;
IF Scans > 2000 THEN
	Test.Fail('the write never finished');
	Run := TRUE;
	RETURN;
END_IF

CASE Phase OF
	0:
		Writer.SetPath(Path);
		Writer.AttachErrorSink(Spy);

		// No RunStarted either, so no document is ever opened.
		Tally.SetLabel('nothing');
		Tally.Begin(0);
		Tally.Finish();
		Writer.RunFinished(Status := Tally, TargetInfo := 'the verifier');
		Phase := 1;
		Run	  := FALSE;

	1:
		Test.AssertTrue(Writer.IsIdle, 'no write was started');
		ExpectedCount := 0;
		ActualCount	  := Writer.FilesWritten;
		Test.AssertEqual(ExpectedCount, ActualCount, 'nothing was written');

		// Not an error either - an empty run is a legitimate deployment.
		ActualCount := Writer.WriteFailures;
		Test.AssertEqual(ExpectedCount, ActualCount, 'and that is not a failure');
		ActualCount := Spy.FrameworkErrorCalls;
		Test.AssertEqual(ExpectedCount, ActualCount, 'and nothing was reported');

		// Now the same run, announced. An empty run IS an outcome and gets a document.
		Writer.RunStarted(Label := 'nothing', TargetInfo := 'a target');
		Writer.RunFinished(Status := Tally, TargetInfo := 'a target');
		Phase := 2;
		Run	  := FALSE;

	2:
		Writer.CyclicLogic();
		IF Writer.IsIdle THEN
			Phase := 3;
		END_IF

		Run := FALSE;

	3:
		ExpectedCount := 1;
		ActualCount	  := Writer.FilesWritten;
		Test.AssertEqual(ExpectedCount, ActualCount, 'an announced empty run does write');
		ExpectedCount := 0;
		ActualCount	  := Writer.WriteFailures;
		Test.AssertEqual(ExpectedCount, ActualCount, 'and not as a failure');
		Run := TRUE;
END_CASE
END_METHOD

END_FUNCTION_BLOCK

// ---- Tests/PureFunctions/TEST_CompareNumericRules.TcPOU
// PORTED from the old verifier. TestValueCompare, numeric rules.

//

// Nothing in the object-level tests pins these: they exercise AssertEqual

// incidentally, which is not the same as pinning what equality MEANS.

//

// Numerics compare BY VALUE across widths - INT#5 equals DINT#5, because the

// storage width is incidental to what the author is checking.

//

// Floats compare EXACTLY. A hidden epsilon inside AssertEqual makes a test passing

// at 1E-7 look identical to one passing exactly; tolerance has its own methods, so

// choosing it is visible at the call site. Because exact float equality is a

// well-known trap, a near miss appends a hint naming those methods - and a hint

// nobody sees is worth nothing, so that is pinned too.
FUNCTION_BLOCK TEST_CompareNumericRules IMPLEMENTS I_Test
VAR
	Result		  : ST_CompareResult;
	SmallFive	  : INT	  := 5;
	BigFive		  : DINT  := 5;
	UnsignedFive  : UDINT := 5;
	Six			  : DINT  := 6;
	OnePointFive  : LREAL := 1.5;
	OnePointFive2 : LREAL := 1.5;
	NearMissA	  : LREAL := 1.0;
	NearMissB	  : LREAL := 1.0000001;
	SumOfTenths	  : LREAL;
	ThreeTenths	  : LREAL	   := 0.3;
	SomeText	  : STRING(20) := 'five';
	ExpectTrue	  : BOOL	   := TRUE;
	ExpectFalse	  : BOOL	   := FALSE;
	ActualEqual	  : BOOL;
	ExpectType	  : E_FailureKind := E_FailureKind.TypeMismatch;
	ActualKind	  : E_FailureKind;
END_VAR

METHOD Run : BOOL
VAR_INPUT
	Enable : BOOL;
	Test   : I_TestAssertions;
END_VAR
// --- value across widths ---------------------------------------------------
Result		:= TestValueCompare(SmallFive, BigFive);
ActualEqual := Result.IsEqual;
Test.AssertEqual(ExpectTrue, ActualEqual, 'INT#5 equals DINT#5');
Result		:= TestValueCompare(SmallFive, UnsignedFive);
ActualEqual := Result.IsEqual;
Test.AssertEqual(ExpectTrue, ActualEqual, 'INT#5 equals UDINT#5');
Result		:= TestValueCompare(BigFive, Six);
ActualEqual := Result.IsEqual;
Test.AssertEqual(ExpectFalse, ActualEqual, '5 does not equal 6');

// --- floats compare exactly ------------------------------------------------
Result		:= TestValueCompare(OnePointFive, OnePointFive2);
ActualEqual := Result.IsEqual;
Test.AssertEqual(ExpectTrue, ActualEqual, 'identical LREALs are equal');

// The canonical binary-floating-point surprise. If a hidden epsilon ever comes

// back, this is what notices.
SumOfTenths := 0.1 + 0.2;
Result		:= TestValueCompare(SumOfTenths, ThreeTenths);
ActualEqual := Result.IsEqual;
Test.AssertEqual(ExpectFalse, ActualEqual, '0.1 + 0.2 does not exactly equal 0.3');

// --- the hint on a near miss -----------------------------------------------
Result := TestValueCompare(NearMissA, NearMissB);
Test.AssertFalse(Result.IsEqual, 'a near miss is still a miss');
Test.AssertTrue(FIND(Result.Diagnostic, 'AssertNear') > 0, 'and the diagnostic names the tolerance methods');

// --- one numeric, one not --------------------------------------------------
Result		:= TestValueCompare(BigFive, SomeText);
ActualEqual := Result.IsEqual;
Test.AssertEqual(ExpectFalse, ActualEqual, 'a number and a string are not equal');
ActualKind := Result.Kind;
Test.AssertEqual(ExpectType, ActualKind, 'and that is a type mismatch, not a value one');
Run := TRUE;
END_METHOD

END_FUNCTION_BLOCK

// ---- Tests/PureFunctions/TEST_CompareTextRules.TcPOU
// TestValueCompare, string rules.

//

// Strings compare by CONTENT. The declared capacity is not the subject - an author

// writing AssertEqual is testing a value, and for a string diSize is the capacity

// of the variable rather than the length of what is in it.

//

// THE WSTRING CASE IS THE ONE THAT MATTERS. Copying WSTRING bytes into a STRING

// buffer and comparing with <> terminates at the first NUL - and every second byte

// of ASCII WSTRING content is NUL, so two different WSTRINGs compare EQUAL and

// tests go green on values that differ. Nothing else in this project would notice

// that happening.
FUNCTION_BLOCK TEST_CompareTextRules IMPLEMENTS I_Test
VAR
	Result		: ST_CompareResult;
	ShortText	: STRING(20)  := 'homed';
	LongText	: STRING(80)  := 'homed';
	OtherText	: STRING(20)  := 'homing';
	WideA		: WSTRING(20) := "homed";
	WideB		: WSTRING(20) := "homer";
	WideC		: WSTRING(20) := "homed";
	ExpectTrue	: BOOL		  := TRUE;
	ExpectFalse : BOOL		  := FALSE;
	ActualEqual : BOOL;
	ExpectNone	: E_FailureKind := E_FailureKind.None;
	ExpectValue : E_FailureKind := E_FailureKind.ValueMismatch;
	ActualKind	: E_FailureKind;
END_VAR

METHOD Run : BOOL
VAR_INPUT
	Enable : BOOL;
	Test   : I_TestAssertions;
END_VAR
// --- capacity is not part of the value -------------------------------------
Result		:= TestValueCompare(ShortText, LongText);
ActualEqual := Result.IsEqual;
Test.AssertEqual(ExpectTrue, ActualEqual, 'STRING(20) and STRING(80) holding the same text are equal');
ActualKind := Result.Kind;
Test.AssertEqual(ExpectNone, ActualKind, 'and carry no failure kind');
Result		:= TestValueCompare(ShortText, OtherText);
ActualEqual := Result.IsEqual;
Test.AssertEqual(ExpectFalse, ActualEqual, 'different text is not equal');

// Same declared size, different content - a VALUE difference, not a size one.
ActualKind := Result.Kind;
Test.AssertEqual(ExpectValue, ActualKind, 'reported as a value difference');

// --- WSTRING is compared AS WSTRING ----------------------------------------

// "homed" and "homer" differ only at the fifth character. Read as a STRING the

// comparison stops at the first NUL - the second byte - and reports equal.
Result		:= TestValueCompare(WideA, WideB);
ActualEqual := Result.IsEqual;
Test.AssertEqual(ExpectFalse, ActualEqual, 'WSTRINGs differing after the first character are not equal');
Result		:= TestValueCompare(WideA, WideC);
ActualEqual := Result.IsEqual;
Test.AssertEqual(ExpectTrue, ActualEqual, 'identical WSTRINGs are equal');

// --- the diagnostic carries both values ------------------------------------
Result := TestValueCompare(ShortText, OtherText);
Test.AssertTrue(FIND(Result.Diagnostic, 'homed') > 0, 'the diagnostic carries expected');
Test.AssertTrue(FIND(Result.Diagnostic, 'homing') > 0, 'and actual');

// And in their own fields, in full - which is what the summary cannot hold.
Test.AssertTrue(FIND(Result.Expected, 'homed') > 0, 'Expected is populated');
Test.AssertTrue(FIND(Result.Actual, 'homing') > 0, 'and so is Actual');
Run := TRUE;
END_METHOD

END_FUNCTION_BLOCK

// ---- Tests/PureFunctions/TEST_CompareOtherRules.TcPOU
// PORTED. TestValueCompare for everything that is neither text nor numeric.

//

// Structs, arrays and enums compare by size and then by bytes. HERE a size

// difference IS a type difference - unlike a string, where capacity is not part of

// the value, two arrays of different length are two different types.
FUNCTION_BLOCK TEST_CompareOtherRules IMPLEMENTS I_Test
VAR
	Result		 : ST_CompareResult;
	RecordA		 : ST_PureSample	   := (Index := 16#6000, SubIndex := 1, Value := 99);
	RecordB		 : ST_PureSample	   := (Index := 16#6000, SubIndex := 1, Value := 99);
	RecordC		 : ST_PureSample	   := (Index := 16#6000, SubIndex := 1, Value := 100);
	ArrayA		 : ARRAY[0..7] OF BYTE := [1, 2, 3, 4, 16#2A, 6, 7, 8];
	ArrayB		 : ARRAY[0..7] OF BYTE := [1, 2, 3, 4, 16#2A, 6, 7, 8];
	ArrayC		 : ARRAY[0..7] OF BYTE := [1, 2, 3, 4, 16#00, 6, 7, 8];
	ArrayShort	 : ARRAY[0..3] OF BYTE := [1, 2, 3, 4];
	ColourRed	 : E_PureColour		   := E_PureColour.Red;
	ColourRedToo : E_PureColour		   := E_PureColour.Red;
	ColourGreen	 : E_PureColour		   := E_PureColour.Green;
	ExpectTrue	 : BOOL				   := TRUE;
	ExpectFalse	 : BOOL				   := FALSE;
	ActualEqual	 : BOOL;
	ExpectType	 : E_FailureKind := E_FailureKind.TypeMismatch;
	ExpectValue	 : E_FailureKind := E_FailureKind.ValueMismatch;
	ActualKind	 : E_FailureKind;
END_VAR

METHOD Run : BOOL
VAR_INPUT
	Enable : BOOL;
	Test   : I_TestAssertions;
END_VAR
// --- structs ---------------------------------------------------------------
Result		:= TestValueCompare(RecordA, RecordB);
ActualEqual := Result.IsEqual;
Test.AssertEqual(ExpectTrue, ActualEqual, 'identical structs are equal');
Result		:= TestValueCompare(RecordA, RecordC);
ActualEqual := Result.IsEqual;
Test.AssertEqual(ExpectFalse, ActualEqual, 'a differing field makes them unequal');
ActualKind := Result.Kind;
Test.AssertEqual(ExpectValue, ActualKind, 'same type, different value');

// --- arrays ----------------------------------------------------------------
Result		:= TestValueCompare(ArrayA, ArrayB);
ActualEqual := Result.IsEqual;
Test.AssertEqual(ExpectTrue, ActualEqual, 'identical arrays are equal');

// They differ at index 4 and nowhere else.
Result := TestValueCompare(ArrayA, ArrayC);
Test.AssertTrue(FIND(Result.Diagnostic, 'byte 4') > 0, 'the diagnostic names the offset of the first difference');
Result		:= TestValueCompare(ArrayA, ArrayShort);
ActualEqual := Result.IsEqual;
Test.AssertEqual(ExpectFalse, ActualEqual, 'arrays of different length are not equal');

// Unlike a string, where capacity is not part of the value.
ActualKind := Result.Kind;
Test.AssertEqual(ExpectType, ActualKind, 'and that is a type mismatch');

// --- enums -----------------------------------------------------------------
Result		:= TestValueCompare(ColourRed, ColourRedToo);
ActualEqual := Result.IsEqual;
Test.AssertEqual(ExpectTrue, ActualEqual, 'identical enum members are equal');
Result		:= TestValueCompare(ColourRed, ColourGreen);
ActualEqual := Result.IsEqual;
Test.AssertEqual(ExpectFalse, ActualEqual, 'different enum members are not equal');
Run := TRUE;
END_METHOD

END_FUNCTION_BLOCK

// ---- Tests/PureFunctions/TEST_SummaryLineComposition.TcPOU
// PORTED. TestSummaryLine.

//

// The composition rule is the part most likely to be got subtly wrong, which is

// why it is a separate pure function rather than logic inside the journal - and

// why it deserves tests of its own rather than being exercised through a verdict.

//

// Order is fixed: step label, then generated diagnostic, then the author's

// message. The author's message is the only element that may be dropped, and it is

// dropped WHOLE - a half sentence leaves the reader unable to tell whether the

// sentence ended or the buffer did, and the full text is in the detail either way.
FUNCTION_BLOCK TEST_SummaryLineComposition IMPLEMENTS I_Test
VAR
	Line		: STRING;
	LongMsg		: T_MaxString;
	LongDiag	: T_MaxString;
	ExpectedLen : INT;
	ActualLen	: INT;
END_VAR

METHOD Run : BOOL
VAR_INPUT
	Enable : BOOL;
	Test   : I_TestAssertions;
END_VAR
// --- the step label leads --------------------------------------------------
Line := TestSummaryLine(StepLabel := 'Home', Diagnostic := 'timed out after 5000 cycles', Message := '');
Test.AssertTrue(FIND(Line, 'Home') = 1, 'the step label leads, because a timeout names its step');

// --- all three, when there is room -----------------------------------------
Line := TestSummaryLine(StepLabel := 'Home', Diagnostic := 'expected 1, actual 2', Message := 'while homing');
Test.AssertTrue(FIND(Line, 'Home') > 0, 'the step label is present');
Test.AssertTrue(FIND(Line, 'expected 1') > 0, 'and the diagnostic');
Test.AssertTrue(FIND(Line, 'while homing') > 0, 'and the author message');

// --- no step label ---------------------------------------------------------
Line := TestSummaryLine(StepLabel := '', Diagnostic := 'expected 1, actual 2', Message := '');
Test.AssertTrue(FIND(Line, 'expected 1') = 1, 'with no step label the diagnostic starts the line');

// --- a message that does not fit is OMITTED, not cut -----------------------
LongMsg := 'this author message is far too long to fit alongside the diagnostic in eighty characters';
Line	:= TestSummaryLine(StepLabel := 'Home', Diagnostic := 'expected 1, actual 2', Message := LongMsg);
Test.AssertTrue(FIND(Line, 'this author message') = 0, 'a message that does not fit is omitted, not truncated');
Test.AssertTrue(FIND(Line, 'expected 1') > 0, 'dropping the message keeps the diagnostic');

// --- the composed line fits ------------------------------------------------
ExpectedLen := 80;
ActualLen	:= LEN(Line);
Test.AssertTrue(ActualLen <= ExpectedLen, 'the composed line fits the summary field');

// --- a diagnostic alone can still overrun, and is marked --------------------
LongDiag  := 'expected a very long rendered value indeed that goes on and on past any reasonable width, actual another one just like it';
Line	  := TestSummaryLine(StepLabel := '', Diagnostic := LongDiag, Message := '');
ActualLen := LEN(Line);
Test.AssertTrue(ActualLen <= ExpectedLen, 'an overlong diagnostic is cut to fit');
Test.AssertTrue(FIND(Line, '...') > 0, 'a cut diagnostic is marked with an ellipsis');
Run := TRUE;
END_METHOD

END_FUNCTION_BLOCK

// ---- Tests/PureFunctions/TEST_ValueRendering.TcPOU
// PORTED. TestValueString and the two type predicates.

//

// Anything unrecognised renders as hex rather than as an empty string. Not

// friendly, but true: a failed comparison of two enums reading 'expected , actual '

// tells the reader nothing at the moment they most need something.
FUNCTION_BLOCK TEST_ValueRendering IMPLEMENTS I_Test
VAR
	Rendered	: T_MaxString;
	SomeDint	: DINT		   := 42;
	SomeReal	: LREAL		   := 1.25;
	SomeText	: STRING(20)   := 'homed';
	SomeWide	: WSTRING(20)  := "wide";
	SomeBool	: BOOL		   := TRUE;
	SomeColour	: E_PureColour := E_PureColour.Green;
	Number		: ST_NumericValue;
	ExpectTrue	: BOOL := TRUE;
	ExpectFalse : BOOL := FALSE;
	ActualFlag	: BOOL;
END_VAR

METHOD Run : BOOL
VAR_INPUT
	Enable : BOOL;
	Test   : I_TestAssertions;
END_VAR
// --- rendering -------------------------------------------------------------
Rendered := TestValueString(SomeDint);
Test.AssertTrue(FIND(Rendered, '42') > 0, 'an integer renders as its digits');
Rendered := TestValueString(SomeReal);
Test.AssertTrue(FIND(Rendered, '1.25') > 0, 'a float renders with its fractional part');
Rendered := TestValueString(SomeText);
Test.AssertTrue(FIND(Rendered, 'homed') > 0, 'a string renders its content');
Rendered := TestValueString(SomeWide);
Test.AssertTrue(FIND(Rendered, 'wide') > 0, 'a WSTRING renders all of its content');
Rendered := TestValueString(SomeBool);
Test.AssertTrue(FIND(Rendered, 'TRUE') > 0, 'a BOOL renders as TRUE or FALSE');

// The case that matters: an unrecognised type class must not render as nothing.
Rendered := TestValueString(SomeColour);
Test.AssertTrue(LEN(Rendered) > 0, 'an enum renders as something rather than nothing');

// --- the predicates --------------------------------------------------------
ActualFlag := TestValueIsText(SomeText);
Test.AssertEqual(ExpectTrue, ActualFlag, 'a STRING is text');
ActualFlag := TestValueIsText(SomeWide);
Test.AssertEqual(ExpectTrue, ActualFlag, 'so is a WSTRING');
ActualFlag := TestValueIsText(SomeDint);
Test.AssertEqual(ExpectFalse, ActualFlag, 'a DINT is not');
ActualFlag := TestValueIsFloat(SomeReal);
Test.AssertEqual(ExpectTrue, ActualFlag, 'an LREAL is a float');
ActualFlag := TestValueIsFloat(SomeDint);
Test.AssertEqual(ExpectFalse, ActualFlag, 'a DINT is not');

// --- numeric conversion ----------------------------------------------------
Number := TestValueAsLReal(SomeDint);
Test.AssertTrue(Number.IsNumeric, 'a DINT converts');
Test.AssertNear(42.0,
				Number.Value,
				0.0001,
				'and keeps its value');

Number := TestValueAsLReal(SomeText);
Test.AssertFalse(Number.IsNumeric, 'a STRING does not convert');
Run := TRUE;
END_METHOD

END_FUNCTION_BLOCK

// ---- Tests/PureFunctions/TEST_ValueBriefShortens.TcPOU
// NEW, not ported - TestValueBrief did not exist in the original.

//

// It is what keeps a composed diagnostic inside CONCAT's 255-character ceiling:

// two full values plus the words between them do not fit, so the summary gets

// shortened copies while the full values travel in their own fields.

//

// The budget is a constant inside the function rather than a parameter, so that

// four call sites cannot carry four copies of the number. That makes the exact

// value an implementation detail - these tests assert the BEHAVIOUR, not the 80.
FUNCTION_BLOCK TEST_ValueBriefShortens IMPLEMENTS I_Test
VAR
	Short		 : T_MaxString := 'homed';
	Long		 : T_MaxString;
	Result		 : T_MaxString;
	Empty		 : T_MaxString := '';
	i			 : DINT;
	ExpectedText : T_MaxString;
	ActualText	 : T_MaxString;
END_VAR

METHOD Run : BOOL
VAR_INPUT
	Enable : BOOL;
	Test   : I_TestAssertions;
END_VAR
// A value comfortably past any sane budget.
Long := '';
FOR i := 1 TO 20 DO
	Long := CONCAT(Long, 'ABCDEFGHIJ');
END_FOR

// --- short values pass through untouched -----------------------------------
ExpectedText := Short;
ActualText	 := TestValueBrief(Short);
Test.AssertEqual(ExpectedText, ActualText, 'a short value is returned unchanged');
ExpectedText := Empty;
ActualText	 := TestValueBrief(Empty);
Test.AssertEqual(ExpectedText, ActualText, 'and so is an empty one');

// --- long values are shortened and marked ----------------------------------
Result := TestValueBrief(Long);
Test.AssertTrue(LEN(Result) < LEN(Long), 'a long value is shortened');
Test.AssertTrue(FIND(Result, '...') > 0, 'and marked with an ellipsis');

// The point of the budget: two of these plus the words between them must still

// fit in a T_MaxString, which CONCAT cannot exceed.
Test.AssertTrue(LEN(Result) <= 100, 'shortened well inside the 255 ceiling');

// The start of the value survives, which is what makes it useful at all.
Test.AssertTrue(FIND(Result, 'ABCDEFGHIJ') = 1, 'the beginning of the value is kept');
Run := TRUE;
END_METHOD

END_FUNCTION_BLOCK

// ---- Tests/Assertions/TEST_AssertNotEqualRejectsSameness.TcPOU
// AssertNotEqual passes when the values DIFFER and fails when they match - which

// is the one thing about it worth checking, because getting it backwards would

// leave every test using it passing on the wrong condition.
FUNCTION_BLOCK TEST_AssertNotEqualRejectsSameness IMPLEMENTS I_Test
VAR
	// A private journal and handle. The assertion under test is driven into THESE,

	// so its verdict can be inspected without the outer suite ever seeing it.
	Subject		  : TestJournal;
	Handle		  : TestVerdict;
	One			  : DINT := 1;
	Two			  : DINT := 2;
	AlsoOne		  : DINT := 1;
	ExpectedCount : UDINT;
	ActualCount	  : UDINT;
END_VAR

METHOD Run : BOOL
VAR_INPUT
	Enable : BOOL;
	Test   : I_TestAssertions;
END_VAR
Handle.Target(Subject);
Subject.Begin('not equal', '');

// Different values: this is the passing case.
Handle.AssertNotEqual(One, Two, 'one is not two');
Test.AssertTrue(Subject.Kind = E_FailureKind.None, 'differing values pass');

// Same values: this must fail.
Handle.AssertNotEqual(One, AlsoOne, 'one IS one');
Test.AssertTrue(Subject.Kind = E_FailureKind.ValueMismatch, 'matching values fail');
ExpectedCount := 2;
ActualCount	  := Subject.AssertionCount;
Test.AssertEqual(ExpectedCount, ActualCount, 'both checks were counted');
Handle.Untarget();
Run := TRUE;
END_METHOD

END_FUNCTION_BLOCK

// ---- Tests/Assertions/TEST_AssertGreaterAndLessCompareTheRightWayRound.TcPOU
// The comparison runs in the direction the name says.

//

// A reversed comparison is the classic defect here, and it is invisible in

// ordinary use: every test written against it simply passes on the wrong

// condition. So both the passing AND the failing direction are checked for each.

//

// Also pinned: a non-ordered type is a TYPE mismatch, not a value one. Comparing a

// string with "greater than" is a mistake in the test, not a finding about the

// code under test.
FUNCTION_BLOCK TEST_AssertGreaterAndLessCompareTheRightWayRound IMPLEMENTS I_Test
VAR
	// A private journal and handle. The assertion under test is driven into THESE,

	// so its verdict can be inspected without the outer suite ever seeing it.
	Subject	 : TestJournal;
	Handle	 : TestVerdict;
	Small	 : DINT		  := 3;
	Large	 : DINT		  := 9;
	SomeText : STRING(20) := 'not a number';
END_VAR

METHOD Run : BOOL
VAR_INPUT
	Enable : BOOL;
	Test   : I_TestAssertions;
END_VAR
Handle.Target(Subject);
Subject.Begin('ordering', '');

// --- AssertGreater ---------------------------------------------------------
Handle.AssertGreater(Large, Small, '9 > 3');
Test.AssertTrue(Subject.Kind = E_FailureKind.None, 'greater passes when it is greater');
Subject.Reset();
Subject.Begin('ordering', '');
Handle.AssertGreater(Small, Large, '3 is not > 9');
Test.AssertTrue(Subject.Kind = E_FailureKind.ValueMismatch, 'and fails when it is not');

// Equal is NOT greater.
Subject.Reset();
Subject.Begin('ordering', '');
Handle.AssertGreater(Small, Small, '3 is not > 3');
Test.AssertTrue(Subject.Kind = E_FailureKind.ValueMismatch, 'equal is not greater');

// --- AssertLess ------------------------------------------------------------
Subject.Reset();
Subject.Begin('ordering', '');
Handle.AssertLess(Small, Large, '3 < 9');
Test.AssertTrue(Subject.Kind = E_FailureKind.None, 'less passes when it is less');
Subject.Reset();
Subject.Begin('ordering', '');
Handle.AssertLess(Large, Small, '9 is not < 3');
Test.AssertTrue(Subject.Kind = E_FailureKind.ValueMismatch, 'and fails when it is not');

// --- a non-ordered type ----------------------------------------------------
Subject.Reset();
Subject.Begin('ordering', '');
Handle.AssertGreater(SomeText, Small, 'a string has no order against a number');
Test.AssertTrue(Subject.Kind = E_FailureKind.TypeMismatch, 'an unordered type is a type mismatch, not a value one');
Handle.Untarget();
Run := TRUE;
END_METHOD

END_FUNCTION_BLOCK

// ---- Tests/Assertions/TEST_AssertNearUsesAbsoluteTolerance.TcPOU
// AssertNear takes tolerance in the UNITS OF THE VALUE - millimetres, volts,

// encoder counts. Its counterpart AssertWithin takes a fraction.

//

// The boundary is what matters. A tolerance that excluded its own edge would make

// every "within 0.1 mm" test subtly stricter than its author intended.
FUNCTION_BLOCK TEST_AssertNearUsesAbsoluteTolerance IMPLEMENTS I_Test
VAR
	// A private journal and handle. The assertion under test is driven into THESE,

	// so its verdict can be inspected without the outer suite ever seeing it.
	Subject : TestJournal;
	Handle	: TestVerdict;
END_VAR

METHOD Run : BOOL
VAR_INPUT
	Enable : BOOL;
	Test   : I_TestAssertions;
END_VAR
Handle.Target(Subject);
Subject.Begin('near', '');

// Inside.
Handle.AssertNear(10.0,
				  10.05,
				  0.1,
				  'well inside');

Test.AssertTrue(Subject.Kind = E_FailureKind.None, 'a value inside the band passes');

// Exactly on the boundary - inclusive.
Subject.Reset();
Subject.Begin('near', '');
Handle.AssertNear(10.0,
				  10.1,
				  0.1,
				  'exactly on the edge');

Test.AssertTrue(Subject.Kind = E_FailureKind.None, 'the boundary itself passes');

// Outside.
Subject.Reset();
Subject.Begin('near', '');
Handle.AssertNear(10.0,
				  10.2,
				  0.1,
				  'outside');

Test.AssertTrue(Subject.Kind = E_FailureKind.ValueMismatch, 'and outside fails');

// The band travels with the expectation, so a reader can see whether the miss

// was meant to pass.

// Summary is composed by Finish, not as checks are recorded - a test with forty

// passing checks composes ONE line, at the end. So the journal is finished before

// its text is read.
Subject.Finish(E_TestStatus.Passed);
Test.AssertTrue(FIND(Subject.Summary, '+/-') > 0, 'the diagnostic names the tolerance, not just the values');

// Symmetric: below the expectation too.
Subject.Reset();
Subject.Begin('near', '');
Handle.AssertNear(10.0,
				  9.8,
				  0.1,
				  'below');

Test.AssertTrue(Subject.Kind = E_FailureKind.ValueMismatch, 'the band is symmetric');
Handle.Untarget();
Run := TRUE;
END_METHOD

END_FUNCTION_BLOCK

// ---- Tests/Assertions/TEST_AssertWithinUsesRelativeTolerance.TcPOU
// AssertWithin takes a FRACTION, so it holds its meaning across magnitudes -

// 0.1 per cent means the same thing at 1.0 and at 1E9, which an absolute tolerance

// does not.

//

// Near zero it collapses to exact equality: the band is a fraction OF the expected

// value, and a fraction of nothing is nothing. That is not a defect to paper over

// with a hidden floor - if zero is the expected value, AssertNear is the method the

// situation calls for, and the diagnostic says so.
FUNCTION_BLOCK TEST_AssertWithinUsesRelativeTolerance IMPLEMENTS I_Test
VAR
	// A private journal and handle. The assertion under test is driven into THESE,

	// so its verdict can be inspected without the outer suite ever seeing it.
	Subject : TestJournal;
	Handle	: TestVerdict;
END_VAR

METHOD Run : BOOL
VAR_INPUT
	Enable : BOOL;
	Test   : I_TestAssertions;
END_VAR
Handle.Target(Subject);
Subject.Begin('within', '');

// 1 per cent of 1000 is 10.
Handle.AssertWithin(1000.0,
					1005.0,
					0.01,
					'inside one per cent');

Test.AssertTrue(Subject.Kind = E_FailureKind.None, 'inside the fraction passes');
Subject.Reset();
Subject.Begin('within', '');
Handle.AssertWithin(1000.0,
					1020.0,
					0.01,
					'outside one per cent');

Test.AssertTrue(Subject.Kind = E_FailureKind.ValueMismatch, 'outside it fails');

// The same FRACTION at a different magnitude - which is the whole point.
Subject.Reset();
Subject.Begin('within', '');
Handle.AssertWithin(0.001,
					0.001005,
					0.01,
					'one per cent of a small number');

Test.AssertTrue(Subject.Kind = E_FailureKind.None, 'the fraction means the same thing at any magnitude');

// Zero: only zero is within any fraction of zero.
Subject.Reset();
Subject.Begin('within', '');
Handle.AssertWithin(0.0,
					0.001,
					0.5,
					'nothing is within half of nothing');

Test.AssertTrue(Subject.Kind = E_FailureKind.ValueMismatch, 'zero admits only zero');

// Summary is composed by Finish, not as checks are recorded - a test with forty

// passing checks composes ONE line, at the end. So the journal is finished before

// its text is read.
Subject.Finish(E_TestStatus.Passed);
Test.AssertTrue(FIND(Subject.Summary, 'AssertNear') > 0, 'and the diagnostic names the method that would work');
Handle.Untarget();
Run := TRUE;
END_METHOD

END_FUNCTION_BLOCK

// ---- Tests/Assertions/TEST_AssertInRangeIsInclusive.TcPOU
// Inclusive on BOTH bounds. A range that excluded its own endpoints would make

// every "between 1 and 10" test mean something narrower than it reads.
FUNCTION_BLOCK TEST_AssertInRangeIsInclusive IMPLEMENTS I_Test
VAR
	// A private journal and handle. The assertion under test is driven into THESE,

	// so its verdict can be inspected without the outer suite ever seeing it.
	Subject : TestJournal;
	Handle	: TestVerdict;
END_VAR

METHOD Run : BOOL
VAR_INPUT
	Enable : BOOL;
	Test   : I_TestAssertions;
END_VAR
Handle.Target(Subject);
Subject.Begin('range', '');
Handle.AssertInRange(5.0,
					 1.0,
					 10.0,
					 'comfortably inside');

Test.AssertTrue(Subject.Kind = E_FailureKind.None, 'inside passes');
Subject.Reset();
Subject.Begin('range', '');
Handle.AssertInRange(1.0,
					 1.0,
					 10.0,
					 'on the lower bound');

Test.AssertTrue(Subject.Kind = E_FailureKind.None, 'the lower bound is included');
Subject.Reset();
Subject.Begin('range', '');
Handle.AssertInRange(10.0,
					 1.0,
					 10.0,
					 'on the upper bound');

Test.AssertTrue(Subject.Kind = E_FailureKind.None, 'and so is the upper');
Subject.Reset();
Subject.Begin('range', '');
Handle.AssertInRange(0.5,
					 1.0,
					 10.0,
					 'below');

Test.AssertTrue(Subject.Kind = E_FailureKind.ValueMismatch, 'below the range fails');
Subject.Reset();
Subject.Begin('range', '');
Handle.AssertInRange(11.0,
					 1.0,
					 10.0,
					 'above');

Test.AssertTrue(Subject.Kind = E_FailureKind.ValueMismatch, 'and above it fails');
Handle.Untarget();
Run := TRUE;
END_METHOD

END_FUNCTION_BLOCK

// ---- Tests/Assertions/TEST_AssertBufferComparisons.TcPOU
// The two pointer comparisons, and the distinction between them.

//

// AssertMemEqual takes ONE length and compares that many bytes. AssertBufferEqual

// takes both lengths and checks them FIRST, so a size difference is reported as a

// SizeMismatch rather than as a difference at whatever byte happens to differ -

// which would send the reader looking at the wrong thing entirely.

//

// A null pointer is Environment, not a value mismatch: nothing was compared, so

// nothing was shown about the code under test.
FUNCTION_BLOCK TEST_AssertBufferComparisons IMPLEMENTS I_Test
VAR
	// A private journal and handle. The assertion under test is driven into THESE,

	// so its verdict can be inspected without the outer suite ever seeing it.
	Subject	 : TestJournal;
	Handle	 : TestVerdict;
	Original : ARRAY[0..7] OF BYTE := [1, 2, 3, 4, 16#2A, 6, 7, 8];
	Copy	 : ARRAY[0..7] OF BYTE := [1, 2, 3, 4, 16#2A, 6, 7, 8];
	Differs	 : ARRAY[0..7] OF BYTE := [1, 2, 3, 4, 16#00, 6, 7, 8];
	Shorter	 : ARRAY[0..3] OF BYTE := [1, 2, 3, 4];
	NoBuffer : POINTER TO BYTE;
END_VAR

METHOD Run : BOOL
VAR_INPUT
	Enable : BOOL;
	Test   : I_TestAssertions;
END_VAR
Handle.Target(Subject);
Subject.Begin('buffers', '');

// --- AssertMemEqual --------------------------------------------------------
Handle.AssertMemEqual(ADR(Original),
					  ADR(Copy),
					  8,
					  'identical buffers');

Test.AssertTrue(Subject.Kind = E_FailureKind.None, 'identical buffers pass');
Subject.Reset();
Subject.Begin('buffers', '');
Handle.AssertMemEqual(ADR(Original),
					  ADR(Differs),
					  8,
					  'differing buffers');

Test.AssertTrue(Subject.Kind = E_FailureKind.ValueMismatch, 'a differing byte fails');

// Summary is composed by Finish, not as checks are recorded - a test with forty

// passing checks composes ONE line, at the end. So the journal is finished before

// its text is read.
Subject.Finish(E_TestStatus.Passed);
Test.AssertTrue(FIND(Subject.Summary, 'byte 4') > 0, 'and the diagnostic names the offset of the first difference');

// A null pointer is not a value finding.
Subject.Reset();
Subject.Begin('buffers', '');
Handle.AssertMemEqual(NoBuffer,
					  ADR(Copy),
					  8,
					  'null expected');

Test.AssertTrue(Subject.Kind = E_FailureKind.Environment, 'a null buffer is environmental, not a mismatch');

// --- AssertBufferEqual: lengths first --------------------------------------
Subject.Reset();
Subject.Begin('buffers', '');
Handle.AssertBufferEqual(ADR(Original),
						 8,
						 ADR(Copy),
						 8,
						 'same length, same content');

Test.AssertTrue(Subject.Kind = E_FailureKind.None, 'equal buffers pass');
Subject.Reset();
Subject.Begin('buffers', '');
Handle.AssertBufferEqual(ADR(Original),
						 8,
						 ADR(Shorter),
						 4,
						 'different lengths');

Test.AssertTrue(Subject.Kind = E_FailureKind.SizeMismatch, 'a length difference is a SIZE mismatch, not a byte one');
Subject.Finish(E_TestStatus.Passed);
Test.AssertTrue(FIND(Subject.Summary, 'bytes') > 0, 'and the summary names both sizes');
Handle.Untarget();
Run := TRUE;
END_METHOD

END_FUNCTION_BLOCK

// ---- Tests/Assertions/TEST_AssertCompletedWithinCountsCompletedScans.TcPOU
// AssertCompletedWithin compares against COMPLETED scans - the one in progress is

// not counted, because the journal is ticked after the body runs.

//

// That is documented in I_TestTiming and is exactly the kind of off-by-one nobody

// notices until a scan budget behaves oddly. Here the journal is ticked by hand so

// the count is unambiguous rather than a side effect of how long something took.
FUNCTION_BLOCK TEST_AssertCompletedWithinCountsCompletedScans IMPLEMENTS I_Test
VAR
	// A private journal and handle. The assertion under test is driven into THESE,

	// so its verdict can be inspected without the outer suite ever seeing it.
	Subject : TestJournal;
	Handle	: TestVerdict;
END_VAR

METHOD Run : BOOL
VAR_INPUT
	Enable : BOOL;
	Test   : I_TestAssertions;
END_VAR
Handle.Target(Subject);
Subject.Begin('budget', '');

// Nothing has completed yet.
Handle.AssertCompletedWithin(2, 'nothing has run');
Test.AssertTrue(Subject.Kind = E_FailureKind.None, 'zero completed scans is within two');

// Two scans completed - still within a budget of two.
Subject.Tick();
Subject.Tick();
Handle.AssertCompletedWithin(2, 'two scans is within two');
Test.AssertTrue(Subject.Kind = E_FailureKind.None, 'the boundary itself passes');

// A third takes it past.
Subject.Tick();
Handle.AssertCompletedWithin(2, 'three scans is not within two');
Test.AssertTrue(Subject.Kind = E_FailureKind.Timeout, 'exceeding the budget is a Timeout, not a value mismatch');

// Summary is composed by Finish, not as checks are recorded - a test with forty

// passing checks composes ONE line, at the end. So the journal is finished before

// its text is read.
Subject.Finish(E_TestStatus.Passed);
Test.AssertTrue(FIND(Subject.Summary, 'cycles') > 0, 'and the summary names cycles');
Handle.Untarget();
Run := TRUE;
END_METHOD

END_FUNCTION_BLOCK

// ---- Tests/PureFunctions/TEST_StopwatchMeasuresAndFreezes.TcPOU
// TestStopwatch. Every duration figure in every report rests on it, and until now

// it is small, old and unglamorous, which is exactly the sort of thing that

// escapes attention.

//

// Resolution is the task period, so a stopwatch read in the same scan it started

// reads zero. That is honest rather than wrong: at this resolution there is nothing

// finer to say, and it is why scan counts are the reproducible measure and elapsed

// time is only reported.
FUNCTION_BLOCK TEST_StopwatchMeasuresAndFreezes IMPLEMENTS I_Test
VAR
	Watch  : TestStopwatch;
	Before : LREAL;
	During : LREAL;
	Frozen : LREAL;
	Again  : LREAL;
	Phase  : DINT;
	Scans  : DINT;
END_VAR

METHOD Run : BOOL
VAR_INPUT
	Enable : BOOL;
	Test   : I_TestAssertions;
END_VAR
Scans := Scans + 1;
IF Scans > 200 THEN
	Test.Fail('the stopwatch never advanced');
	Run := TRUE;
	RETURN;
END_IF

CASE Phase OF
	0:
		Test.AssertFalse(Watch.IsRunning, 'a fresh stopwatch is not running');
		Before := Watch.Elapsed;
		Test.AssertTrue(Before = 0.0, 'and reads zero');
		Watch.Start();
		Test.AssertTrue(Watch.IsRunning, 'and is running once started');
		Phase := 1;
		Run	  := FALSE;

	1:
		// Let real scans pass. Nothing else can make this advance.
		IF Scans > 20 THEN
			During := Watch.Elapsed;
			Phase  := 2;
		END_IF

		Run := FALSE;

	2:
		Test.AssertTrue(During > 0.0, 'it advances while running');
		Frozen := Watch.Stop();
		Test.AssertFalse(Watch.IsRunning, 'and stops when stopped');
		Test.AssertTrue(Frozen > 0.0, 'Stop returns what it measured');
		Phase := 3;
		Run	  := FALSE;

	3:
		IF Scans > 40 THEN
			Again := Watch.Elapsed;
			Phase := 4;
		END_IF

		Run := FALSE;

	4:
		// The whole point of stopping: a test that finished twenty scans ago must not
		// keep accruing time while the suite runs the next one.
		Test.AssertTrue(Again = Frozen, 'a stopped stopwatch does not keep advancing');

		// Stopping twice returns what it held rather than zero.
		Test.AssertTrue(Watch.Stop() = Frozen, 'and stopping again returns the same value');
		Watch.Reset();
		Test.AssertTrue(Watch.Elapsed = 0.0, 'Reset clears it');
		Test.AssertFalse(Watch.IsRunning, 'and leaves it stopped');
		Run := TRUE;
END_CASE

Run := TRUE;
END_METHOD

END_FUNCTION_BLOCK

// ---- Tests/Suite/TEST_RegisteredAndReporterCountsAreReadable.TcPOU
// The two counts Plan.md tells CI to assert, and which nothing had ever read.

//

// They exist for the same hazard: a test or a sink that silently stops being

// registered takes its output with it, and the run simply comes out smaller. CI

// sees fewer passes rather than a failure, which reads as an improvement.
FUNCTION_BLOCK TEST_RegisteredAndReporterCountsAreReadable IMPLEMENTS I_Test
VAR
	Runner		  : TestRun<2>;
	Suite		  : TestSuite<4>;
	SpyOne		  : SpyReporter;
	SpyTwo		  : SpyReporter;
	A			  : PassingTest;
	B			  : PassingTest;
	Budgets		  : ST_TestBudgets;
	ExpectedCount : UDINT;
	ActualCount	  : UDINT;
END_VAR

METHOD Run : BOOL
VAR_INPUT
	Enable : BOOL;
	Test   : I_TestAssertions;
END_VAR
Suite.SetLabel('inner');
Suite.Register(A, 'first', Budgets);
Suite.Register(B, 'second', Budgets);
ExpectedCount := 2;
ActualCount	  := Suite.RegisteredCount;
Test.AssertEqual(ExpectedCount, ActualCount, 'the suite counts what it registered');
Runner.SetLabel('a run');
Runner.AddReporter(SpyOne);
Runner.AddReporter(SpyTwo);
Runner.AddSuite(Suite);
ActualCount := Runner.ReporterCount;
Test.AssertEqual(ExpectedCount, ActualCount, 'the run counts its sinks');

// Pushed into the suite as well, which is the one attachment point working.
ActualCount := Suite.ReporterCount;
Test.AssertEqual(ExpectedCount, ActualCount, 'and the suite received them');
ExpectedCount := 1;
ActualCount	  := Runner.SuiteCount;
Test.AssertEqual(ExpectedCount, ActualCount, 'and the run counts its suites');
Run := TRUE;
END_METHOD

END_FUNCTION_BLOCK

// ---- Tests/Watchdog/TEST_WatchdogAbandonsAStalledSuite.TcPOU
// A suite that stops progressing is named, counted and left behind, rather than

// holding the run open forever.

//

// A suite cannot detect this about itself - it IS the thing that has stopped - so

// the run, which owns the sequence, is the only object positioned to notice.
FUNCTION_BLOCK TEST_WatchdogAbandonsAStalledSuite IMPLEMENTS I_Test
VAR
	Runner		  : TestRun<2>;
	Stalled		  : StallingSuite;
	Recorder	  : RecordingReporter;
	Phase		  : DINT;
	Scans		  : DINT;
	ExpectedCount : UDINT;
	ActualCount	  : UDINT;
END_VAR

METHOD Run : BOOL
VAR_INPUT
	Enable : BOOL;
	Test   : I_TestAssertions;
END_VAR
Scans := Scans + 1;
IF Scans > 500 THEN
	// The watchdog itself failing to fire looks exactly like the run hanging, which
	// is why this guard exists rather than trusting it.
	Test.Fail('the watchdog never fired');
	Run := TRUE;
	RETURN;
END_IF

CASE Phase OF
	0:
		Runner.SetLabel('a run');
		Runner.AddReporter(Recorder);
		Runner.AddSuite(Stalled);

		// Small, so the test is cheap. The default is generous because it is a backstop

		// and a legitimately slow suite must not trip it.
		Runner.SetWatchdog(20);
		Phase := 1;
		Run	  := FALSE;

	1:
		IF Runner.Run(Enable := TRUE) THEN
			Phase := 2;
		END_IF

		Run := FALSE;

	2:
		Test.AssertTrue(Runner.IsComplete, 'the run completed rather than hanging');
		ExpectedCount := 1;
		ActualCount	  := Runner.StalledSuites;
		Test.AssertEqual(ExpectedCount, ActualCount, 'one suite was abandoned');

		// One call with Enable FALSE, and its return ignored.
		ActualCount := Stalled.AbandonCalls;
		Test.AssertEqual(ExpectedCount, ActualCount, 'abandoned with exactly one call');

		// Named, so a reader knows WHICH suite stopped.
		Test.AssertTrue(Recorder.ErrorCount > 0, 'the stall was reported');
		Test.AssertTrue(Recorder.ErrorContains('a stalled suite'), 'and the report names the suite');

		// A stall is a framework error, never a test failure - nothing about the code

		// under test was shown.
		Test.AssertTrue(Runner.Outcome = E_RunOutcome.Errored, 'and the run cannot be trusted');
		Run := TRUE;
END_CASE
END_METHOD

END_FUNCTION_BLOCK

// ---- Doubles/StallingSuite.TcPOU
// A suite that never completes and never brings a test to a verdict.

//

// The only failure the suite watchdog exists to catch. Per-test deadlines already

// bound every test that did not disable them, so what is left is a framework

// defect or a test that turned its own deadlines off - and from outside, both look

// exactly like this.

//

// Implements I_TestSuite, which is I_TestExecution plus I_TestRunStatus. It does

// not implement I_TestConfiguration, so a run pushing reporters into it finds

// nothing through __QUERYINTERFACE and moves on - which is worth exercising too.
FUNCTION_BLOCK StallingSuite IMPLEMENTS I_TestSuite
VAR
	_RunCalls	  : UDINT;
	_AbandonCalls : UDINT;
	_PassedCount  : UDINT;
	_Skipped	  : BOOL;
END_VAR

// Exactly 1 after the watchdog fires, however many scans the run has left.
PROPERTY AbandonCalls : UDINT
GET
AbandonCalls := _AbandonCalls;
END_GET
END_PROPERTY

// Bring one test to a verdict, so a test can prove the watchdog measures PROGRESS

// and not elapsed time: a suite that keeps completing tests is never abandoned,

// however long it takes.
METHOD CompleteOneTest
_PassedCount := _PassedCount + 1;
END_METHOD

PROPERTY ErrorCount : UDINT
GET
ErrorCount := 0;
END_GET
END_PROPERTY

PROPERTY FailedCount : UDINT
GET
FailedCount := 0;
END_GET
END_PROPERTY

PROPERTY IsComplete : BOOL
GET
IsComplete := FALSE;
END_GET
END_PROPERTY

PROPERTY Label : T_MaxString
GET
Label := 'a stalled suite';
END_GET
END_PROPERTY

PROPERTY Outcome : E_RunOutcome
GET
Outcome := E_RunOutcome.Running;
END_GET
END_PROPERTY

PROPERTY PassedCount : UDINT
GET
PassedCount := _PassedCount;
END_GET
END_PROPERTY

// Never finishes, and never brings a test to a verdict. The only thing the

// watchdog can catch.
METHOD Run : BOOL
VAR_INPUT
	Enable : BOOL;
END_VAR
IF NOT Enable THEN
	// The abandon call. Counted so a test can prove the run made exactly one.
	_AbandonCalls := _AbandonCalls + 1;

	// Deliberately does NOT report itself finished. A suite that has stopped will

	// not answer this either, and the run must not wait for it.
	Run := FALSE;
	RETURN;
END_IF

_RunCalls := _RunCalls + 1;
Run		  := FALSE;
END_METHOD

PROPERTY RunCalls : UDINT
GET
RunCalls := _RunCalls;
END_GET
END_PROPERTY

METHOD Skip
_Skipped := TRUE;
END_METHOD

PROPERTY SkippedCount : UDINT
GET
SkippedCount := 0;
END_GET
END_PROPERTY

PROPERTY TestCount : UDINT
GET
TestCount := 2;
END_GET
END_PROPERTY

PROPERTY TotalDuration : LREAL
GET
TotalDuration := 0.0;
END_GET
END_PROPERTY

END_FUNCTION_BLOCK

// ---- Tests/Watchdog/TEST_WatchdogMeasuresProgressNotTime.TcPOU
// The measure is VERDICTS REACHED, not scans elapsed.

//

// A rig suite waiting on hardware can sit for minutes and be perfectly healthy -

// it still finishes its tests one at a time. Counting scans since the suite

// STARTED would abandon the slow along with the stuck, which would make the

// watchdog worse than not having one.

//

// Here the suite completes a test every few scans and never finishes. It must run

// far past its own watchdog budget untouched.
FUNCTION_BLOCK TEST_WatchdogMeasuresProgressNotTime IMPLEMENTS I_Test
VAR
	Runner		  : TestRun<2>;
	Slow		  : StallingSuite;
	Recorder	  : RecordingReporter;
	Phase		  : DINT;
	Scans		  : DINT;
	Ticks		  : DINT;
	ExpectedCount : UDINT;
	ActualCount	  : UDINT;
END_VAR

METHOD Run : BOOL
VAR_INPUT
	Enable : BOOL;
	Test   : I_TestAssertions;
END_VAR
Scans := Scans + 1;
CASE Phase OF
	0:
		Runner.SetLabel('a run');
		Runner.AddReporter(Recorder);
		Runner.AddSuite(Slow);
		Runner.SetWatchdog(10);
		Phase := 1;
		Run	  := FALSE;

	1:
		// Well past 10 scans in total, but never 10 WITHOUT a verdict.
		Runner.Run(Enable := TRUE);
		Ticks := Ticks + 1;
		IF (Ticks MOD 5) = 0 THEN
			Slow.CompleteOneTest();
		END_IF

		IF Ticks >= 60 THEN
			Phase := 2;
		END_IF

		Run := FALSE;

	2:
		// Sixty scans against a ten-scan budget, and still running.
		ExpectedCount := 0;
		ActualCount	  := Runner.StalledSuites;
		Test.AssertEqual(ExpectedCount, ActualCount, 'a progressing suite is never abandoned');
		ActualCount := Slow.AbandonCalls;
		Test.AssertEqual(ExpectedCount, ActualCount, 'and was never asked to stop');
		ActualCount := Recorder.ErrorCount;
		Test.AssertEqual(ExpectedCount, ActualCount, 'and nothing was reported');
		Test.AssertFalse(Runner.IsComplete, 'the run is still going, as it should be');
		Run := TRUE;
END_CASE
END_METHOD

END_FUNCTION_BLOCK

// ---- Tests/Watchdog/TEST_WatchdogZeroDisablesIt.TcPOU
// Zero disables, as every other deadline in this library does.

//

// For a rig where a single test legitimately outlasts any sane budget and the

// operator would rather wait than be second-guessed.
FUNCTION_BLOCK TEST_WatchdogZeroDisablesIt IMPLEMENTS I_Test
VAR
	Runner		  : TestRun<2>;
	Stalled		  : StallingSuite;
	Recorder	  : RecordingReporter;
	Phase		  : DINT;
	Ticks		  : DINT;
	ExpectedCount : UDINT;
	ActualCount	  : UDINT;
END_VAR

METHOD Run : BOOL
VAR_INPUT
	Enable : BOOL;
	Test   : I_TestAssertions;
END_VAR
CASE Phase OF
	0:
		Runner.SetLabel('a run');
		Runner.AddReporter(Recorder);
		Runner.AddSuite(Stalled);
		Runner.SetWatchdog(0);
		Phase := 1;
		Run	  := FALSE;

	1:
		Runner.Run(Enable := TRUE);
		Ticks := Ticks + 1;
		IF Ticks >= 100 THEN
			Phase := 2;
		END_IF

		Run := FALSE;

	2:
		// A hundred scans with no progress at all, and untouched.
		ExpectedCount := 0;
		ActualCount	  := Runner.StalledSuites;
		Test.AssertEqual(ExpectedCount, ActualCount, 'a zero budget never fires');
		ActualCount := Stalled.AbandonCalls;
		Test.AssertEqual(ExpectedCount, ActualCount, 'and nothing was abandoned');
		Test.AssertFalse(Runner.IsComplete, 'the run waits, which is what was asked for');
		Run := TRUE;
END_CASE
END_METHOD

END_FUNCTION_BLOCK

// ---- Tests/Characterization/CHAR_Capacity.TcPOU
// Part of the acceptance contract: behaviour a project depending on this library

// is entitled to rely on.

//

// Two things. CAPACITY HOLDS WHAT IT SAYS - a TestSuite<3> takes three tests and

// refuses the fourth. And OVERFLOW IS REPORTED rather than suppressed: the run

// still finishes and the result document is still written, because a missing

// artifact reads to CI as a broken pipeline rather than as a rejected test.

//

// The refusal is a FRAMEWORK ERROR, not a testcase. Registration is explicit, so a

// rejected test is refused at the call and never becomes a case - but it is never

// silent, which is the part that matters.
FUNCTION_BLOCK CHAR_Capacity IMPLEMENTS I_Test
VAR
	Inner	 : TestSuite<3>;
	Recorder : RecordingReporter;

	// A run, not just a suite. RunFinished is a run-level event and only a TestRun

	// raises it - which is what produces a result document at all. Without one, a

	// single-suite project writes nothing, and this test is what found that.
	Runner		  : TestRun<2>;
	Budgets		  : ST_TestBudgets;
	Phase		  : DINT;
	Scans		  : DINT;
	A			  : PassingTest;
	B			  : PassingTest;
	C			  : PassingTest;
	D			  : PassingTest;
	AcceptedA	  : BOOL;
	AcceptedB	  : BOOL;
	AcceptedC	  : BOOL;
	AcceptedD	  : BOOL;
	ExpectedCount : UDINT;
	ActualCount	  : UDINT;
END_VAR

METHOD Run : BOOL
VAR_INPUT
	Enable : BOOL;
	Test   : I_TestAssertions;
END_VAR
Scans := Scans + 1;
IF Scans > 500 THEN
	Test.Fail('the inner suite never completed');
	Run := TRUE;
	RETURN;
END_IF

CASE Phase OF
	0:
		Inner.SetLabel('CHAR_Capacity_Subject');
		Runner.SetLabel('CHAR_Capacity_Subject_Run');

		// Attached to the RUN, which pushes it into every suite. One attachment point.
		Runner.AddReporter(Recorder);
		Runner.AddSuite(Inner);
		AcceptedA := Inner.Register(A, 'A', Budgets);
		AcceptedB := Inner.Register(B, 'B', Budgets);
		AcceptedC := Inner.Register(C, 'C', Budgets);

		// One too many.
		AcceptedD := Inner.Register(D, 'D', Budgets);
		Phase	  := 1;
		Run		  := FALSE;

	1:
		IF Runner.Run(Enable := TRUE) THEN
			Phase := 2;
		END_IF

		Run := FALSE;

	2:
		Test.AssertTrue(AcceptedA, 'the first fits');
		Test.AssertTrue(AcceptedB, 'the second fits');
		Test.AssertTrue(AcceptedC, 'three tests fit a TestSuite<3>');
		Test.AssertFalse(AcceptedD, 'the fourth overflows');

		// Never silent.
		Test.AssertTrue(Recorder.ErrorCount > 0, 'the overflow was reported');
		Test.AssertTrue(Recorder.ErrorContains('D'), 'and named the test it refused');
		ExpectedCount := 3;
		ActualCount	  := Recorder.CaseCount;
		Test.AssertEqual(ExpectedCount, ActualCount, 'three cases were recorded');

		// Overflow must not suppress the artifact.
		ExpectedCount := 1;
		ActualCount	  := Recorder.SaveCount;
		Test.AssertEqual(ExpectedCount, ActualCount, 'and the document was still written');
		Run := TRUE;
END_CASE
END_METHOD

END_FUNCTION_BLOCK

// ---- Tests/Characterization/CHAR_OverflowStatistics.TcPOU
// Part of the acceptance contract: the Errors figure is distinct from Failures.

//

// An overflow is a framework error, not a failed assertion. Conflating them sends

// whoever reads the report hunting a defect that is not there. Three tests

// registered and passing, one refused, and the statistics say exactly that - and

// the result document is still written.
FUNCTION_BLOCK CHAR_OverflowStatistics IMPLEMENTS I_Test
VAR
	Inner	 : TestSuite<3>;
	Recorder : RecordingReporter;

	// A run, not just a suite. RunFinished is a run-level event and only a TestRun

	// raises it - which is what produces a result document at all. Without one, a

	// single-suite project writes nothing, and this test is what found that.
	Runner		  : TestRun<2>;
	Budgets		  : ST_TestBudgets;
	Phase		  : DINT;
	Scans		  : DINT;
	A			  : PassingTest;
	B			  : PassingTest;
	C			  : PassingTest;
	D			  : PassingTest;
	ExpectedCount : UDINT;
	ActualCount	  : UDINT;
END_VAR

METHOD Run : BOOL
VAR_INPUT
	Enable : BOOL;
	Test   : I_TestAssertions;
END_VAR
Scans := Scans + 1;
IF Scans > 500 THEN
	Test.Fail('the inner suite never completed');
	Run := TRUE;
	RETURN;
END_IF

CASE Phase OF
	0:
		Inner.SetLabel('CHAR_Overflow_Subject');
		Runner.SetLabel('CHAR_Overflow_Subject_Run');

		// Attached to the RUN, which pushes it into every suite. One attachment point.
		Runner.AddReporter(Recorder);
		Runner.AddSuite(Inner);
		Inner.Register(A, 'A', Budgets);
		Inner.Register(B, 'B', Budgets);
		Inner.Register(C, 'C', Budgets);
		Inner.Register(D, 'D', Budgets);
		Phase := 1;
		Run	  := FALSE;

	1:
		IF Runner.Run(Enable := TRUE) THEN
			Phase := 2;
		END_IF

		Run := FALSE;

	2:
		ExpectedCount := 3;
		ActualCount	  := Recorder.StatTests;
		Test.AssertEqual(ExpectedCount, ActualCount, 'three tests registered');
		ExpectedCount := 1;
		ActualCount	  := Recorder.StatErrors;
		Test.AssertEqual(ExpectedCount, ActualCount, 'overflow counted as an error');
		ExpectedCount := 0;
		ActualCount	  := Recorder.StatFailures;
		Test.AssertEqual(ExpectedCount, ActualCount, 'and not as a failure');
		ExpectedCount := 1;
		ActualCount	  := Recorder.SaveCount;
		Test.AssertEqual(ExpectedCount, ActualCount, 'the result document was still written');
		Run := TRUE;
END_CASE
END_METHOD

END_FUNCTION_BLOCK

// ---- Tests/Characterization/CHAR_ReRunTests.TcPOU
// PORTED. The assertion that matters most is the suite-node count.

//

// A defect in this library's history had the reset loop appending one testsuite

// node per array element to the existing document - five nodes per re-run for a

// suite declared <4>, not one. Counting them is how a reintroduction gets caught,

// and nothing else in the verifier counts them.

//

// Also pinned: a re-run produces a fresh document and a second save, and every

// test really runs again.
FUNCTION_BLOCK CHAR_ReRunTests IMPLEMENTS I_Test
VAR
	Inner	 : TestSuite<4>;
	Recorder : RecordingReporter;

	// A run, not just a suite. The DOCUMENT boundary belongs to the run, so a

	// re-run that is to produce a fresh artifact has to be re-run at this level.
	Runner			: TestRun<2>;
	Budgets			: ST_TestBudgets;
	Phase			: DINT;
	Scans			: DINT;
	X				: PassingTest;
	Y				: PassingTest;
	CasesAfterRun1	: UDINT;
	SuitesAfterRun1 : UDINT;
	ExpectedCount	: UDINT;
	ActualCount		: UDINT;
END_VAR

METHOD Run : BOOL
VAR_INPUT
	Enable : BOOL;
	Test   : I_TestAssertions;
END_VAR
Scans := Scans + 1;
IF Scans > 500 THEN
	Test.Fail('the inner suite never completed');
	Run := TRUE;
	RETURN;
END_IF

CASE Phase OF
	0:
		Inner.SetLabel('CHAR_ReRun_Subject');
		Inner.Register(X, 'X', Budgets);
		Inner.Register(Y, 'Y', Budgets);
		Runner.SetLabel('CHAR_ReRun_Run');
		Runner.AddReporter(Recorder);
		Runner.AddSuite(Inner);
		Phase := 1;
		Run	  := FALSE;

	1:
		IF Runner.Run(Enable := TRUE) THEN
			CasesAfterRun1	:= Recorder.CaseCount;
			SuitesAfterRun1 := Recorder.SuiteCount;

			// At the RUN, not the suite. Re-running the suite alone re-executes its

			// tests but announces no run, so no second document is produced.
			Runner.ReRun();
			Phase := 2;
		END_IF

		Run := FALSE;

	2:
		IF Runner.Run(Enable := TRUE) THEN
			Phase := 3;
		END_IF

		Run := FALSE;

	3:
		ExpectedCount := 2;
		ActualCount	  := CasesAfterRun1;
		Test.AssertEqual(ExpectedCount, ActualCount, 'two cases in the first run');
		ExpectedCount := 1;
		ActualCount	  := SuitesAfterRun1;
		Test.AssertEqual(ExpectedCount, ActualCount, 'one suite node in the first run');
		ExpectedCount := 4;
		ActualCount	  := Recorder.CaseCount;
		Test.AssertEqual(ExpectedCount, ActualCount, 'two more cases after the re-run');

		// The one that catches the historical defect.
		ExpectedCount := 2;
		ActualCount	  := Recorder.SuiteCount;
		Test.AssertEqual(ExpectedCount, ActualCount, 'exactly one suite node per run');
		ActualCount := Recorder.SaveCount;
		Test.AssertEqual(ExpectedCount, ActualCount, 'the re-run produced a second document');

		// And the tests really ran twice, rather than the counts being replayed.
		ActualCount := X.BodyCalls;
		Test.AssertEqual(ExpectedCount, ActualCount, 'the first test ran twice');
		Run := TRUE;
END_CASE
END_METHOD

END_FUNCTION_BLOCK

// ---- Tests/Characterization/CHAR_ReRunIndividual.TcPOU
// PORTED. An individual re-run is a debugging aid and must NOT touch the result

// document - letting it append would corrupt the CI artifact with duplicate

// entries.

//

// Three things, all of which must hold: the test really did run

// again, no new case was recorded, and no new document was produced. Without the

// first, the test would pass even if ReRunSingle did nothing at all.
FUNCTION_BLOCK CHAR_ReRunIndividual IMPLEMENTS I_Test
VAR
	Inner		   : TestSuite<4>;
	Recorder	   : RecordingReporter;
	Budgets		   : ST_TestBudgets;
	Phase		   : DINT;
	Scans		   : DINT;
	X			   : PassingTest;
	Y			   : PassingTest;
	Accepted	   : BOOL;
	CasesAfterRun1 : UDINT;
	SavesAfterRun1 : UDINT;
	ExpectedCount  : UDINT;
	ActualCount	   : UDINT;
END_VAR

METHOD Run : BOOL
VAR_INPUT
	Enable : BOOL;
	Test   : I_TestAssertions;
END_VAR
Scans := Scans + 1;
IF Scans > 500 THEN
	Test.Fail('the inner suite never completed');
	Run := TRUE;
	RETURN;
END_IF

CASE Phase OF
	0:
		Inner.SetLabel('CHAR_Individual_Subject');
		Inner.AddReporter(Recorder);
		Inner.Register(X, 'X', Budgets);
		Inner.Register(Y, 'Y', Budgets);
		Phase := 1;
		Run	  := FALSE;

	1:
		IF Inner.Run(Enable := TRUE) THEN
			CasesAfterRun1 := Recorder.CaseCount;
			SavesAfterRun1 := Recorder.SaveCount;
			Accepted	   := Inner.ReRunSingle('X');
			Phase		   := 2;
		END_IF

		Run := FALSE;

	2:
		IF Inner.Run(Enable := TRUE) THEN
			Phase := 3;
		END_IF

		Run := FALSE;

	3:
		Test.AssertTrue(Accepted, 'the individual re-run was accepted');

		// It really ran. Without this the rest would pass on a no-op.
		ExpectedCount := 2;
		ActualCount	  := X.BodyCalls;
		Test.AssertEqual(ExpectedCount, ActualCount, 'the chosen test really re-ran');
		ExpectedCount := 1;
		ActualCount	  := Y.BodyCalls;
		Test.AssertEqual(ExpectedCount, ActualCount, 'and nothing else did');

		// And recorded nothing.
		ExpectedCount := CasesAfterRun1;
		ActualCount	  := Recorder.CaseCount;
		Test.AssertEqual(ExpectedCount, ActualCount, 'the re-run recorded no new case');
		ExpectedCount := SavesAfterRun1;
		ActualCount	  := Recorder.SaveCount;
		Test.AssertEqual(ExpectedCount, ActualCount, 'and produced no new document');
		Run := TRUE;
END_CASE
END_METHOD

END_FUNCTION_BLOCK

// ---- Tests/Characterization/CHAR_WallClockTimeout.TcPOU
// Part of the acceptance contract: the wall-clock deadline fires, and says so.

//

// The scan budget is the easier one to reach for and the easier one to test, so

// this is the deadline most likely to go unexercised.

//

// The inner test never finishes, so only a deadline can end it. Its CYCLE budget

// is set to zero so the wall clock is unambiguously what fired; without that, at a

// fast task period a cycle budget could expire first and the test would pass for

// the wrong reason.

//

// The second assertion is the one that matters: the failure must NAME the wall

// clock. A deadline that fires correctly but says the wrong thing is still a

// defect - the message is what someone reads at three in the morning.
FUNCTION_BLOCK CHAR_WallClockTimeout IMPLEMENTS I_Test
VAR
	Inner		  : TestSuite<4>;
	Recorder	  : RecordingReporter;
	Budgets		  : ST_TestBudgets;
	Phase		  : DINT;
	Scans		  : DINT;
	Spinner		  : HangingBodyTest;
	ExpectedCount : UDINT;
	ActualCount	  : UDINT;
END_VAR

METHOD Run : BOOL
VAR_INPUT
	Enable : BOOL;
	Test   : I_TestAssertions;
END_VAR
Scans := Scans + 1;
IF Scans > 500 THEN
	Test.Fail('the inner suite never completed');
	Run := TRUE;
	RETURN;
END_IF

CASE Phase OF
	0:
		// Zero disables the scan budget. Explicitly SET, not merely left alone - an
		// unset field inherits the suite default instead of disabling anything.
		Budgets.Body.Cycles		  := 0;
		Budgets.Body.IsCyclesSet  := TRUE;
		Budgets.Body.Timeout	  := T#200MS;
		Budgets.Body.IsTimeoutSet := TRUE;
		Inner.SetLabel('CHAR_WallClock_Subject');
		Inner.AddReporter(Recorder);
		Inner.Register(Spinner, 'Spinner', Budgets);
		Phase := 1;
		Run	  := FALSE;

	1:
		IF Inner.Run(Enable := TRUE) THEN
			Phase := 2;
		END_IF

		Run := FALSE;

	2:
		ExpectedCount := 1;
		ActualCount	  := Recorder.StatFailures;
		Test.AssertEqual(ExpectedCount, ActualCount, 'the spinning test failed');
		Test.AssertTrue(Recorder.CaseFailureKind('Spinner') = E_FailureKind.Timeout, 'and failed as a timeout');
		Test.AssertTrue(Recorder.FailureContains('Spinner', 'wall time'), 'the failure names the wall-clock deadline');
		Run := TRUE;
END_CASE
END_METHOD

END_FUNCTION_BLOCK

// ---- Tests/Characterization/CHAR_TimeoutPrecedence.TcPOU
// PORTED. Three rules, one inner test each, none of which ever finishes - so only

// a deadline can end them:

//

//   DefaultCycles     claims nothing      -> the suite default applies

//   OverrideCycles    claims cycles       -> the per-test value wins

//   OverrideTimeOnly  claims wall clock   -> wall clock overridden, but the

//                                            suite's CYCLE budget still applies

//

// The third is the subtle one and the reason this test exists. Overrides are

// tracked separately per unit, so naming one does not silently disable the other.

// A single "overridden" flag would break exactly this case and nothing else would

// notice.

//

// The suite default is five cycles, so the whole test costs about thirty.
FUNCTION_BLOCK CHAR_TimeoutPrecedence IMPLEMENTS I_Test
VAR
	Inner			 : TestSuite<4>;
	Recorder		 : RecordingReporter;
	Budgets			 : ST_TestBudgets;
	Phase			 : DINT;
	Scans			 : DINT;
	DefaultCycles	 : HangingBodyTest;
	OverrideCycles	 : HangingBodyTest;
	OverrideTimeOnly : HangingBodyTest;
	Defaults		 : ST_TestBudgets;
	OwnCycles		 : ST_TestBudgets;
	OwnTimeOnly		 : ST_TestBudgets;
	ExpectedCount	 : UDINT;
	ActualCount		 : UDINT;
END_VAR

METHOD Run : BOOL
VAR_INPUT
	Enable : BOOL;
	Test   : I_TestAssertions;
END_VAR
Scans := Scans + 1;
IF Scans > 500 THEN
	Test.Fail('the inner suite never completed');
	Run := TRUE;
	RETURN;
END_IF

